// TwinCAT 3 PLC project PLC_InjectionMolding
// ProgramVersion: 3.1.4024.0
// libraries:
//   Tc2_Standard, * (Beckhoff Automation GmbH)
//   Tc2_System, * (Beckhoff Automation GmbH)
//   Tc3_Module, * (Beckhoff Automation GmbH)
//   Tc3_Vision, * (Beckhoff Automation GmbH)
//   VisuDialogs, * (System)
// project tree:
//   DUTs/ ST_ProductionData.TcDUT, E_AlarmID.TcDUT, E_MachineMode.TcDUT, E_SequenceState.TcDUT, ST_Recipe.TcDUT, ST_VisionResult.TcDUT
//   / GlobalTextList.TcGTLO, PlcTask.TcTTO, Visualization Manager.TcVMO (not stored)
//   GVLs/ GVL_Config.TcGVL, GVL_IO.TcGVL, GVL_Simulation.TcGVL, GVL_Status.TcGVL
//   POUs/ FB_AlarmManager.TcPOU, FB_AnalogInput.TcPOU, FB_Extruder.TcPOU, FB_Hopper.TcPOU, FB_InjectionSequence.TcPOU, FB_Interlocks.TcPOU, FB_Machine.TcPOU, FB_Mold.TcPOU, FB_PlantSimulation.TcPOU, FB_TemperatureControl.TcPOU, FB_Vision.TcPOU, MAIN.TcPOU, PRG_VisionTest.TcPOU
//   VISUs/ Visualization_Overview.TcVIS
// real-time tasks:
//   TASK PlcTask: cycle T#10ms, priority 20, ADS port 350

CONFIGURATION PLC_InjectionMolding
    RESOURCE PLC ON TwinCAT3
        TASK PlcTask(INTERVAL := T#10ms, PRIORITY := 20);
        PROGRAM MAIN WITH PlcTask : MAIN;
        PROGRAM PRG_VisionTest WITH PlcTask : PRG_VisionTest;
    END_RESOURCE
END_CONFIGURATION

// ---- DUTs/ST_ProductionData.TcDUT
TYPE ST_ProductionData :
STRUCT
	nTotalParts        : UDINT;
    nGoodParts         : UDINT;
    nRejectedParts     : UDINT;

    fRejectRate        : REAL;

    tLastCycleTime     : TIME;

    nLastDefectCode    : UINT;
	
	fLastCycleTimeSec : REAL;
END_STRUCT
END_TYPE

// ---- DUTs/E_AlarmID.TcDUT
{attribute 'qualified_only'}
{attribute 'strict'}
TYPE E_AlarmID :
(
	ALARM_NONE:=0,
	
	//HOPPER
	ALARM_HOPPER_LOW_TIMEOUT:=1001,
	ALARM_HOPPER_FILL_TIMEOUT:=1002,
	
	//TEMPERATURE/PRESSURE
	ALARM_TEMP_LOW:=2001,
	ALARM_TEMP_HIGH:=2002,
	ALARM_PRESSURE_HIGH:=2003,
	
	//MOLD/MOTION
	ALARM_MOLD_OPEN_TIMEOUT:=3001,
	ALARM_MOLD_CLOSE_TIMEOUT:=3002,
	
	//VISION
	ALARM_VISION_OFFLINE:=4001,
	ALARM_VISION_TIMEOUT:=4002,
	
	//SAFETY
	ALARM_GUARD_OPEN:=9001,
	ALARM_ESTOP:=9002
);
END_TYPE

// ---- DUTs/E_MachineMode.TcDUT
{attribute 'qualified_only'}
{attribute 'strict'}
TYPE E_MachineMode :
(
	MODE_INITIAL := 0,
    MODE_STARTUP := 1,
    MODE_STOPPED := 2,
    MODE_RUN := 3,
    MODE_SHUTDOWN := 4,
    MODE_ESTOP := 5	
);
END_TYPE

// ---- DUTs/E_SequenceState.TcDUT
{attribute 'qualified_only'}
{attribute 'strict'}
TYPE E_SequenceState :
(
	SEQ_IDLE :=0,
	SEQ_INJECT :=1,
	SEQ_COOLING :=2,
	SEQ_DOSING :=3,
	SEQ_OPEN_MOLD :=4,
	SEQ_EJECT:=5,
	SEQ_CLOSE_MOLD:=6,
	
	//Vision
	SEQ_VISION_TRIGGER:=7,
	SEQ_VISION_WAIT:=8,
	SEQ_SORT_PART:=9,
	
	SEQ_COMPLETE:= 10
);
END_TYPE

// ---- DUTs/ST_Recipe.TcDUT
TYPE ST_Recipe :
STRUCT
	sProductName		: STRING(40);
	
	fBarrelTempSP       : REAL;
    fPressureLimit      : REAL;

    tCoolingTime        : TIME;
    tInjectionTimeout   : TIME;

    nVisionJob          : UINT;

    fWidthMin           : REAL;
    fWidthMax           : REAL;
    fHeightMin          : REAL;
    fHeightMax          : REAL;
	
END_STRUCT
END_TYPE

// ---- DUTs/ST_VisionResult.TcDUT
TYPE ST_VisionResult :
STRUCT

    // Vision system status
    bReady       : BOOL;
    bBusy        : BOOL;

    // Result handshake
    bResultValid : BOOL;

    // Inspection result
    bPartPresent : BOOL;
    bPartOK      : BOOL;

    // Classification
    nDefectCode  : UINT;

    // Measured geometry
    // Currently stored in pixels
    fWidth       : REAL;
    fHeight      : REAL;
    fAngle       : REAL;

    // Identification of inspected part
    nProductID   : DINT;

END_STRUCT
END_TYPE

// ---- GVLs/GVL_Config.TcGVL
{attribute 'qualified_only'}
VAR_GLOBAL
	// Temperature Configuration
	
	c_fStartupTempSP      : REAL := 120.0;
    c_fShutdownTempSP     : REAL := 20.0;
    c_fShutdownComplete   : REAL := 30.0;
	
	// Pressure Limits
	
	c_fStartupPressure    : REAL := 4.0;
    c_fMaxPressure        : REAL := 100.0;
	c_fMinOperatingTemp	  : REAL := 80.0;
	
	// Process Timing
	
	c_tCoolingTime        : TIME := T#5S;
	
	// Hopper Monitoring
	
	c_tHopperLowTimeout   : TIME := T#30S;
    c_tHopperFillTimeout  : TIME := T#180S;
	
	// Production
	
	c_nBatchSize          : UDINT := 1000;	
	
END_VAR

// ---- GVLs/GVL_IO.TcGVL
{attribute 'qualified_only'}
VAR_GLOBAL
	
	//Operator Inputs
	
	B_start		: BOOL;
	B_ES		: BOOL;
	B_ack		: BOOL;
	B_startup	: BOOL;
	B_shutdown	: BOOL;
	B_stop		: BOOL;
	
	//Position Sensors
	
	ES101		: BOOL;
	ES102		: BOOL;
	ES201		: BOOL;
	ES202		: BOOL;
	
	//Safety
	
	S101		: BOOL;
	
	//Hopper Sensors
	
	LIS101		: BOOL;
	LIS102		: BOOL;	
	
	//Analog Inputs
	
	PI101_raw	: INT;
	TI101_raw	: INT;
	TI201_raw	: INT;
	
	//Motors
	
	M101         : BOOL;
    M102         : BOOL;
    M201_l       : BOOL;
    M201_r       : BOOL;
    M301         : BOOL;
	
	//Valves
	
	V1           : BOOL;
    V2           : BOOL;
    V3           : BOOL;
	
	//Heating
	
	P_in		 : REAL;
	
	//Hopper Warning
	
	W_hopper	 : BOOL;
	
END_VAR

// ---- GVLs/GVL_Simulation.TcGVL
{attribute 'qualified_only'}

VAR_GLOBAL

    // =====================================================
    // MASTER SWITCH
    // =====================================================

    bSimulationEnabled : BOOL := TRUE;


    // =====================================================
    // FAULT INJECTION
    // =====================================================

    bForcePressureHigh : BOOL := FALSE;
    bForceTempLow      : BOOL := FALSE;

    bForceES101Fault   : BOOL := FALSE;
    bForceES102Fault   : BOOL := FALSE;
    bForceES201Fault   : BOOL := FALSE;
    bForceES202Fault   : BOOL := FALSE;

    bForceLIS101Fault  : BOOL := FALSE;
    bForceLIS102Fault  : BOOL := FALSE;


    // =====================================================
    // VISION FAULT INJECTION
    // =====================================================

    bForceVisionOffline : BOOL := FALSE;

    // Kept for compatibility / old commissioning logic.
    // The new FB_Vision does not need this for real defect detection.
    bForceVisionReject  : BOOL := FALSE;

    bForceVisionTimeout : BOOL := FALSE;


    // =====================================================
    // VISION IMAGE SOURCE
    // =====================================================

    // Used by FB_Vision.
    // In manual mode, set this directly.
    // In random mode, MAIN updates it automatically.
    sVisionImagePath : STRING(255) :=
        'C:\TcVision\good_reference.png';


    // =====================================================
    // RANDOM VIRTUAL PART MODE
    // =====================================================

    // FALSE = manually choose sVisionImagePath
    // TRUE  = randomly select one dataset image
    //         whenever a new part enters SEQ_INJECT
    bRandomPartMode : BOOL := TRUE;


    // Current image selected for the molded part
    nVisionDatasetIndex : INT := 1;


    // Seed for pseudo-random number generator
    // Fixed value makes the sequence reproducible
    nRandomSeed : UDINT := 123456789;


    // =====================================================
    // RANDOM VISION DATASET
    // =====================================================

    aVisionDataset : ARRAY[1..40] OF STRING(255) := [

        'C:\TcVision\RandomDataset\part_001.png',
        'C:\TcVision\RandomDataset\part_002.png',
        'C:\TcVision\RandomDataset\part_003.png',
        'C:\TcVision\RandomDataset\part_004.png',
        'C:\TcVision\RandomDataset\part_005.png',
        'C:\TcVision\RandomDataset\part_006.png',
        'C:\TcVision\RandomDataset\part_007.png',
        'C:\TcVision\RandomDataset\part_008.png',
        'C:\TcVision\RandomDataset\part_009.png',
        'C:\TcVision\RandomDataset\part_010.png',

        'C:\TcVision\RandomDataset\part_011.png',
        'C:\TcVision\RandomDataset\part_012.png',
        'C:\TcVision\RandomDataset\part_013.png',
        'C:\TcVision\RandomDataset\part_014.png',
        'C:\TcVision\RandomDataset\part_015.png',
        'C:\TcVision\RandomDataset\part_016.png',
        'C:\TcVision\RandomDataset\part_017.png',
        'C:\TcVision\RandomDataset\part_018.png',
        'C:\TcVision\RandomDataset\part_019.png',
        'C:\TcVision\RandomDataset\part_020.png',

        'C:\TcVision\RandomDataset\part_021.png',
        'C:\TcVision\RandomDataset\part_022.png',
        'C:\TcVision\RandomDataset\part_023.png',
        'C:\TcVision\RandomDataset\part_024.png',
        'C:\TcVision\RandomDataset\part_025.png',
        'C:\TcVision\RandomDataset\part_026.png',
        'C:\TcVision\RandomDataset\part_027.png',
        'C:\TcVision\RandomDataset\part_028.png',
        'C:\TcVision\RandomDataset\part_029.png',
        'C:\TcVision\RandomDataset\part_030.png',

        'C:\TcVision\RandomDataset\part_031.png',
        'C:\TcVision\RandomDataset\part_032.png',
        'C:\TcVision\RandomDataset\part_033.png',
        'C:\TcVision\RandomDataset\part_034.png',
        'C:\TcVision\RandomDataset\part_035.png',
        'C:\TcVision\RandomDataset\part_036.png',
        'C:\TcVision\RandomDataset\part_037.png',
        'C:\TcVision\RandomDataset\part_038.png',
        'C:\TcVision\RandomDataset\part_039.png',
        'C:\TcVision\RandomDataset\part_040.png'

    ];

END_VAR

// ---- GVLs/GVL_Status.TcGVL
{attribute 'qualified_only'}
VAR_GLOBAL
	

	eMachineMode:
		E_MachineMode:= E_MachineMode.MODE_INITIAL;
		
	eSequenceState:
		E_SequenceState:= E_SequenceState.SEQ_IDLE;
		
	stProduction:
		ST_ProductionData;
		
	stVision:
		ST_VisionResult;
		
	//Process Values
	
	fPressureBar      : REAL := 0.0;
    fBarrelTemp       : REAL := 20.0;
    fMoldTemp         : REAL := 20.0;

	//Machine Status

	bMachineReady     : BOOL := FALSE;
    bCycleActive      : BOOL := FALSE;
    bFaultActive      : BOOL := FALSE;	
	
	eActiveAlarm : E_AlarmID := E_AlarmID.ALARM_NONE;
	sSequenceText : STRING(32) := 'IDLE';
	sMachineModeText : STRING(20) := 'INITIAL';
	sActiveAlarmText : STRING(40) := 'NONE';
END_VAR

// ---- POUs/MAIN.TcPOU
PROGRAM MAIN
VAR
	fbPlantSim   : FB_PlantSimulation;

    fbPressure   : FB_AnalogInput;
    fbBarrelTemp : FB_AnalogInput;
    fbMoldTemp   : FB_AnalogInput;
	fbMachine	 : FB_Machine;
	fbTemperature: FB_TemperatureControl;
	fbInjectionSequence : FB_InjectionSequence;
	fbExtruder	 : FB_Extruder;
	fbMold		 : FB_Mold;
	fbHopper	 : FB_Hopper;
	fbAlarmManager : FB_AlarmManager;
	fbInterlocks : FB_Interlocks;

	// Temporary manual commands for commissioning/testing
	bTestM101_Request   : BOOL := FALSE;
	bTestM102_Request   : BOOL := FALSE;
	bTestM201_l_Request : BOOL := FALSE;
	bTestM201_r_Request : BOOL := FALSE;
	
	 // Vision
    fbVision              : FB_Vision;
    bVisionTestTrigger    : BOOL := FALSE;
    bVisionTestAck        : BOOL := FALSE;
    nVisionTestProductID  : DINT := 1;
    bVisionOffline        : BOOL := FALSE;
	bVisionTimeout : BOOL;
	
	
	nRandomValue : UDINT;
	
	ePreviousSequenceState : E_SequenceState := E_SequenceState.SEQ_IDLE;
	
END_VAR

										// ANALOG INPUT PROCESSING


// Pressure PI101: 0 ... 200 bar
fbPressure(
    nRaw := GVL_IO.PI101_raw,
    fEngMin := 0.0,
    fEngMax := 200.0,
    fValue => GVL_Status.fPressureBar
);


// Barrel temperature TI101: -100 ... 600 °C
fbBarrelTemp(
    nRaw := GVL_IO.TI101_raw,
    fEngMin := -100.0,
    fEngMax := 600.0,
    fValue => GVL_Status.fBarrelTemp
);


// Mold temperature TI201: -100 ... 600 °C
fbMoldTemp(
    nRaw := GVL_IO.TI201_raw,
    fEngMin := -100.0,
    fEngMax := 600.0,
    fValue => GVL_Status.fMoldTemp
);

														// MACHINE MODE CONTROL

fbMachine(
    bStartup := GVL_IO.B_startup,
    bStart := GVL_IO.B_start,
    bStop := GVL_IO.B_stop,
    bShutdown := GVL_IO.B_shutdown,
    bEStop := GVL_IO.B_ES,
    bAck := GVL_IO.B_ack,

    fBarrelTemp := GVL_Status.fBarrelTemp,
    fPressureBar := GVL_Status.fPressureBar,
    bMoldClosed := GVL_IO.ES202,

    bSequenceStopComplete :=
        fbInjectionSequence.bStopComplete,

    eMode => GVL_Status.eMachineMode,
    bMachineReady => GVL_Status.bMachineReady,

    bV2 => GVL_IO.V2,
    bV3 => GVL_IO.V3
);


														// TEMPERATURE CONTROL
fbTemperature(
    bEnable := fbMachine.bTempControlEnable,
	fSetpoint := fbMachine.fTempSetpoint,
    fActualTemp := GVL_Status.fBarrelTemp,

    fHeatingPower => GVL_IO.P_in,
    bCoolingValve => GVL_IO.V1
);

													// AUTOMATIC INJECTION SEQUENCE


fbInjectionSequence(
    bEnable :=
        GVL_Status.eMachineMode =
        E_MachineMode.MODE_RUN,

    bStopRequest := GVL_IO.B_stop,

    bAtFront := GVL_IO.ES101,
    bAtRear := GVL_IO.ES102,

    bMoldOpen := GVL_IO.ES201,
    bMoldClosed := GVL_IO.ES202,

    tCoolingTime := GVL_Config.c_tCoolingTime,

    nProducedParts :=
        GVL_Status.stProduction.nTotalParts,

    nBatchSize :=
        GVL_Config.c_nBatchSize,
		
	bVisionReady :=
    	GVL_Status.stVision.bReady,

	bVisionResultValid :=
    	GVL_Status.stVision.bResultValid,

	bVisionPartOK :=
    	GVL_Status.stVision.bPartOK,
		
	bVisionOffline := fbVision.bOffline,

	bVisionTimeout := fbVision.bTimeout,

    eState => GVL_Status.eSequenceState,
	
	tLastCycleTime =>
        GVL_Status.stProduction.tLastCycleTime
);

	GVL_Status.bCycleActive := fbInjectionSequence.bCycleActive;
	
	GVL_Status.stProduction.fLastCycleTimeSec :=
    	TIME_TO_REAL(GVL_Status.stProduction.tLastCycleTime) / 1000.0;
	

CASE GVL_Status.eMachineMode OF

    E_MachineMode.MODE_INITIAL:
        GVL_Status.sMachineModeText := 'INITIAL';

    E_MachineMode.MODE_STARTUP:
        GVL_Status.sMachineModeText := 'STARTUP';

    E_MachineMode.MODE_STOPPED:
        GVL_Status.sMachineModeText := 'STOPPED';

    E_MachineMode.MODE_RUN:
        GVL_Status.sMachineModeText := 'RUN';

    E_MachineMode.MODE_SHUTDOWN:
        GVL_Status.sMachineModeText := 'SHUTDOWN';

    E_MachineMode.MODE_ESTOP:
        GVL_Status.sMachineModeText := 'E-STOP';

ELSE
    GVL_Status.sMachineModeText := 'UNKNOWN';

END_CASE;





CASE fbInjectionSequence.eState OF

    E_SequenceState.SEQ_IDLE:
        GVL_Status.sSequenceText := 'IDLE';

    E_SequenceState.SEQ_INJECT:
        GVL_Status.sSequenceText := 'INJECT';

    E_SequenceState.SEQ_COOLING:
        GVL_Status.sSequenceText := 'COOLING';

    E_SequenceState.SEQ_DOSING:
        GVL_Status.sSequenceText := 'DOSING';

    E_SequenceState.SEQ_OPEN_MOLD:
        GVL_Status.sSequenceText := 'OPEN MOLD';

    E_SequenceState.SEQ_EJECT:
        GVL_Status.sSequenceText := 'EJECT';

    E_SequenceState.SEQ_CLOSE_MOLD:
        GVL_Status.sSequenceText := 'CLOSE MOLD';

    E_SequenceState.SEQ_VISION_TRIGGER:
        GVL_Status.sSequenceText := 'VISION TRIGGER';

    E_SequenceState.SEQ_VISION_WAIT:
        GVL_Status.sSequenceText := 'VISION WAIT';

    E_SequenceState.SEQ_SORT_PART:
        GVL_Status.sSequenceText := 'SORT PART';

    E_SequenceState.SEQ_COMPLETE:
        GVL_Status.sSequenceText := 'COMPLETE';

ELSE
    GVL_Status.sSequenceText := 'UNKNOWN';

END_CASE;



// =====================================================
// RANDOM VIRTUAL PART GENERATOR
// Select exactly one image when a new cycle enters
// SEQ_INJECT.
// =====================================================

IF GVL_Simulation.bRandomPartMode
   AND
   (fbInjectionSequence.eState = E_SequenceState.SEQ_INJECT)
   AND
   (ePreviousSequenceState <> E_SequenceState.SEQ_INJECT) THEN

    // -------------------------------------------------
    // Generate next pseudo-random number
    // -------------------------------------------------

    GVL_Simulation.nRandomSeed :=
        (GVL_Simulation.nRandomSeed * UDINT#1664525)
        + UDINT#1013904223;

    nRandomValue :=
        GVL_Simulation.nRandomSeed;


    // -------------------------------------------------
    // Map pseudo-random value to dataset index 1..40
    // -------------------------------------------------

    GVL_Simulation.nVisionDatasetIndex :=
        UDINT_TO_INT(
            nRandomValue MOD UDINT#40
        ) + 1;


    // -------------------------------------------------
    // Assign selected image to this molded part
    // -------------------------------------------------

    GVL_Simulation.sVisionImagePath :=
        GVL_Simulation.aVisionDataset[
            GVL_Simulation.nVisionDatasetIndex
        ];

END_IF;


// =====================================================
// STORE CURRENT STATE FOR NEXT PLC SCAN
// This line MUST come after the random-selection logic.
// =====================================================

ePreviousSequenceState :=
    fbInjectionSequence.eState;	
	
	
	
	
											// COUNT PRODUCED PARTS

IF fbInjectionSequence.bPartCompleted THEN

    GVL_Status.stProduction.nTotalParts :=
        GVL_Status.stProduction.nTotalParts + 1;

END_IF;

// Good part counter
IF fbInjectionSequence.bGoodPart THEN

    GVL_Status.stProduction.nGoodParts :=
        GVL_Status.stProduction.nGoodParts + 1;

END_IF;


// Rejected part counter
IF fbInjectionSequence.bRejectedPart THEN

    GVL_Status.stProduction.nRejectedParts :=
        GVL_Status.stProduction.nRejectedParts + 1;

    // Store meaningful reject reason
    IF fbVision.bOffline THEN

        // Vision system unavailable
        GVL_Status.stProduction.nLastDefectCode := UINT#4001;

    ELSIF fbVision.bTimeout THEN

        // Vision inspection timeout
        GVL_Status.stProduction.nLastDefectCode := UINT#4002;

    ELSE

        // Genuine Cognex / simulated inspection defect
        GVL_Status.stProduction.nLastDefectCode :=
            GVL_Status.stVision.nDefectCode;

    END_IF;

END_IF;


// Reject rate
IF GVL_Status.stProduction.nTotalParts > 0 THEN

    GVL_Status.stProduction.fRejectRate :=
        (
            UDINT_TO_REAL(
                GVL_Status.stProduction.nRejectedParts
            )
            /
            UDINT_TO_REAL(
                GVL_Status.stProduction.nTotalParts
            )
        ) * 100.0;

ELSE

    GVL_Status.stProduction.fRejectRate := 0.0;

END_IF;


											// EQUIPMENT CONTROL (Extruder + MOLD)

fbExtruder(
    bRotateCmd :=
        fbMachine.bStartupRotateCmd
        OR fbInjectionSequence.bRotateCmd,

    bInjectCmd :=
        fbInjectionSequence.bInjectCmd,

    bES101 := GVL_IO.ES101,
    bES102 := GVL_IO.ES102
);

fbMold(
    bOpenCmd :=
        fbInjectionSequence.bOpenMoldCmd,

    bCloseCmd :=
        fbMachine.bStartupCloseCmd
        OR fbInjectionSequence.bCloseMoldCmd,

    bES201 := GVL_IO.ES201,
    bES202 := GVL_IO.ES202
);

										// MACHINE INTERLOCKS

fbInterlocks(
    eMode := GVL_Status.eMachineMode,
	bM101_Request := fbExtruder.bRotateRequest,
    bM102_Request := fbExtruder.bInjectRequest,
    bM201_l_Request := fbMold.bOpenRequest,
    bM201_r_Request := fbMold.bCloseRequest,

    bES101 := GVL_IO.ES101,
    bES102 := GVL_IO.ES102,
    bES201 := GVL_IO.ES201,
    bES202 := GVL_IO.ES202,

    bGuardOpen := GVL_IO.S101,

    fPressureBar := GVL_Status.fPressureBar,
    fBarrelTemp := GVL_Status.fBarrelTemp,

    bM101_Enable => GVL_IO.M101,
    bM102_Enable => GVL_IO.M102,
    bM201_l_Enable => GVL_IO.M201_l,
    bM201_r_Enable => GVL_IO.M201_r
);

																	// HOPPER CONTROL

fbHopper(
    eMode := GVL_Status.eMachineMode,

    bLIS101 := GVL_IO.LIS101,
    bLIS102 := GVL_IO.LIS102,

    bAck := GVL_IO.B_ack,

    bFeederRequest => GVL_IO.M301,
    bWarning => GVL_IO.W_hopper
);


// =====================================================
// RANDOM VIRTUAL PART GENERATOR
// Select one image exactly once when entering SEQ_INJECT
// =====================================================

IF GVL_Simulation.bRandomPartMode
   AND
   (fbInjectionSequence.eState = E_SequenceState.SEQ_INJECT)
   AND
   (ePreviousSequenceState <> E_SequenceState.SEQ_INJECT) THEN

    // Generate next pseudo-random number
    GVL_Simulation.nRandomSeed :=
        (GVL_Simulation.nRandomSeed * UDINT#1664525)
        + UDINT#1013904223;

    nRandomValue :=
        GVL_Simulation.nRandomSeed;


    // Convert random value to dataset index 1..40
    GVL_Simulation.nVisionDatasetIndex :=
        UDINT_TO_INT(
            nRandomValue MOD UDINT#40
        ) + 1;


    // Assign selected image to current molded part
    GVL_Simulation.sVisionImagePath :=
        GVL_Simulation.aVisionDataset[
            GVL_Simulation.nVisionDatasetIndex
        ];

END_IF;


// IMPORTANT:
// Store current state only AFTER the random selection check
ePreviousSequenceState :=
    fbInjectionSequence.eState;



																	// VISION SYSTEM
// Temporary simulation / commissioning interface

fbVision(
    bEnable :=
        (GVL_Status.eMachineMode = E_MachineMode.MODE_RUN),

    bTrigger :=
        fbInjectionSequence.bVisionTrigger,

    bAck :=
        fbInjectionSequence.bVisionAck,

    bFaultAck :=
        GVL_IO.B_ack,

    bForceOffline :=
        GVL_Simulation.bForceVisionOffline,

    bForceTimeout :=
        GVL_Simulation.bForceVisionTimeout,

    nProductID :=
        UDINT_TO_DINT(
            GVL_Status.stProduction.nTotalParts + 1
        ),
		
	sImagePath :=
		GVL_Simulation.sVisionImagePath,

    stResult =>
        GVL_Status.stVision,

    bOffline =>
        bVisionOffline,
		
	bTimeout =>
        bVisionTimeout
);

																	// ALARM MANAGEMENT


fbAlarmManager(
    eMode := GVL_Status.eMachineMode,

    bHopperLowTimeout :=
        fbHopper.bLowLevelTimeout,

    bHopperFillTimeout :=
        fbHopper.bFillTimeout,

    fBarrelTemp :=
        GVL_Status.fBarrelTemp,

    fPressureBar :=
        GVL_Status.fPressureBar,

    bGuardOpen :=
        GVL_IO.S101,

    bEStop :=
        GVL_IO.B_ES,

    bVisionOffline :=
        bVisionOffline,

    bVisionTimeout :=
		fbVision.bTimeout,

    bAck :=
        GVL_IO.B_ack,

    bFaultActive =>
        GVL_Status.bFaultActive,

    eActiveAlarm =>
        GVL_Status.eActiveAlarm
);

CASE GVL_Status.eActiveAlarm OF

    E_AlarmID.ALARM_NONE:
        GVL_Status.sActiveAlarmText := 'NONE';

    E_AlarmID.ALARM_VISION_OFFLINE:
        GVL_Status.sActiveAlarmText := 'VISION OFFLINE';

    E_AlarmID.ALARM_VISION_TIMEOUT:
        GVL_Status.sActiveAlarmText := 'VISION TIMEOUT';

ELSE
    GVL_Status.sActiveAlarmText := 'ALARM ACTIVE';

END_CASE;

											// PLANT SIMULATION

fbPlantSim(
    bEnable := GVL_Simulation.bSimulationEnabled,

    bM101 := GVL_IO.M101,
    bM102 := GVL_IO.M102,
    bM201_l := GVL_IO.M201_l,
    bM201_r := GVL_IO.M201_r,
    bM301 := GVL_IO.M301,

    bV1 := GVL_IO.V1,
    bV2 := GVL_IO.V2,
    bV3 := GVL_IO.V3,

    fHeaterPower := GVL_IO.P_in,

    eMode := GVL_Status.eMachineMode,

    bES101 => GVL_IO.ES101,
    bES102 => GVL_IO.ES102,
    bES201 => GVL_IO.ES201,
    bES202 => GVL_IO.ES202,

    bLIS101 => GVL_IO.LIS101,
    bLIS102 => GVL_IO.LIS102,

    nPI101Raw => GVL_IO.PI101_raw,
    nTI101Raw => GVL_IO.TI101_raw,
    nTI201Raw => GVL_IO.TI201_raw
);

//PRG_VisionTest();

END_PROGRAM

// ---- POUs/FB_PlantSimulation.TcPOU
FUNCTION_BLOCK FB_PlantSimulation
VAR_INPUT
	bEnable		: BOOL;
	
	//Motors
	
	bM101		: BOOL;
	bM102		: BOOL;
	bM201_l		: BOOL;
	bM201_r		: BOOL;
	bM301		: BOOL;
	
	// Valves
	bV1			: BOOL;
	bV2			: BOOL;
	bV3			: BOOL;
	
	// Heater
	fHeaterPower: REAL;
	
	//machine Operating Mode
	eMode		: E_MachineMode;	
END_VAR
VAR_OUTPUT
	// Screw end switches
    bES101        : BOOL;
    bES102        : BOOL;

    // Mold end switches
    bES201        : BOOL;
    bES202        : BOOL;

    // Hopper level switches
    bLIS101       : BOOL;
    bLIS102       : BOOL;

    // Simulated analog inputs
    nPI101Raw     : INT;
    nTI101Raw     : INT;
    nTI201Raw     : INT;
END_VAR
VAR
	 // Positions: 0 ... 100 %
    fScrewPosition : REAL := 50.0;
    fMoldPosition  : REAL := 0.0;
    fHopperLevel   : REAL := 75.0;

    // Physical process values
    fPressure      : REAL := 0.0;
    fBarrelTemp    : REAL := 20.0;
    fMoldTemp      : REAL := 20.0;
END_VAR

IF bEnable THEN

    									// Injection screw simulation

    // Injection cylinder pushes screw forward
    IF bM102 THEN
        fScrewPosition := fScrewPosition + 1.0;
    END_IF;


    // During normal operation M101 performs dosing,
    // causing the screw to move backwards.
    IF bM101 AND
       (eMode = E_MachineMode.MODE_RUN) THEN

        fScrewPosition := fScrewPosition - 0.5;

    END_IF;


    // Limit screw position
    fScrewPosition :=
        LIMIT(0.0, fScrewPosition, 100.0);


    // Generate end switches
    bES101 := (fScrewPosition >= 100.0);
    bES102 := (fScrewPosition <= 0.0);



   
    											// Mold simulation
  

    IF bM201_l THEN
        fMoldPosition := fMoldPosition - 0.2;
    END_IF;

    IF bM201_r THEN
        fMoldPosition := fMoldPosition + 0.2;
    END_IF;


    fMoldPosition :=
        LIMIT(0.0, fMoldPosition, 100.0);


    bES201 := (fMoldPosition <= 0.0);
    bES202 := (fMoldPosition >= 100.0);

	
    										 // Hopper simulation
											 

    IF bM301 THEN

        fHopperLevel := fHopperLevel + 0.05;

    ELSIF eMode = E_MachineMode.MODE_RUN THEN

        // Material consumption
        fHopperLevel := fHopperLevel - 0.002;

    END_IF;


    fHopperLevel :=
        LIMIT(0.0, fHopperLevel, 100.0);


    // Low-level sensor
    //bLIS101 := (fHopperLevel > 20.0);

    // High-level sensor
    //bLIS102 := (fHopperLevel >= 90.0);
	
	// Normal level-switch simulation
	bLIS101 := (fHopperLevel > 20.0);
	bLIS102 := (fHopperLevel >= 90.0);

	// Fault injection
	IF GVL_Simulation.bForceLIS101Fault THEN
    	bLIS101 := FALSE;
	END_IF;

	IF GVL_Simulation.bForceLIS102Fault THEN
    	bLIS102 := FALSE;
	END_IF;



    									// Barrel Temperature Simulation

    IF fHeaterPower > 0.0 THEN

        fBarrelTemp :=
            fBarrelTemp +
            (fHeaterPower / 100.0) * 0.03;

    END_IF;


    // Cooling valve
    IF bV1 THEN
        fBarrelTemp := fBarrelTemp - 0.02;
    END_IF;


    // Natural cooling toward ambient
    IF (fHeaterPower <= 0.0) AND NOT bV1 THEN

        IF fBarrelTemp > 20.0 THEN
            fBarrelTemp := fBarrelTemp - 0.002;
        END_IF;

    END_IF;


    fBarrelTemp :=
        LIMIT(-100.0, fBarrelTemp, 600.0);


										   // Mold Temperature Simulation

    IF bV2 OR bV3 THEN

        IF fMoldTemp > 20.0 THEN
            fMoldTemp := fMoldTemp - 0.01;
        END_IF;

    END_IF;


    fMoldTemp :=
        LIMIT(-100.0, fMoldTemp, 600.0);


										    // Pressure Simulation
 

// During startup, screw rotation fills the nozzle
// and pressure gradually rises.
IF eMode = E_MachineMode.MODE_STARTUP THEN

    IF bM101 THEN
        fPressure := fPressure + 0.01;
    END_IF;


// During normal production
ELSIF eMode = E_MachineMode.MODE_RUN THEN

    // Injection temporarily raises pressure
    IF bM102 THEN

        fPressure := fPressure + 0.10;

    ELSE

        // Pressure relaxes after injection
        IF fPressure > 5.0 THEN
            fPressure := fPressure - 0.10;

        ELSIF fPressure < 5.0 THEN
            fPressure := fPressure + 0.01;
        END_IF;

    END_IF;


// Machine not producing
ELSE

    IF fPressure > 0.0 THEN
        fPressure := fPressure - 0.05;
    END_IF;

END_IF;


// Physical limits
fPressure :=
    LIMIT(0.0, fPressure, 200.0);

						    // Convert physical values back to raw PLC signals
 
    nPI101Raw :=
        REAL_TO_INT(
            (fPressure / 200.0) * 32767.0
        );


    nTI101Raw :=
        REAL_TO_INT(
            ((fBarrelTemp + 100.0) / 700.0)
            * 32767.0
        );


    nTI201Raw :=
        REAL_TO_INT(
            ((fMoldTemp + 100.0) / 700.0)
            * 32767.0
        );

END_IF;

END_FUNCTION_BLOCK

// ---- POUs/FB_AnalogInput.TcPOU
FUNCTION_BLOCK FB_AnalogInput
VAR_INPUT
	nRaw	:	INT;
	fEngMin :	REAL;
	fEngMax :	REAL;
END_VAR

VAR_OUTPUT
	fValue  :	REAL;
	bValid  :	BOOL;
END_VAR

VAR
	fRaw	:	REAL;
END_VAR

fRaw:= INT_TO_REAL(nRaw);

bValid := (nRaw >= 0);

IF bValid THEN
	fValue := fEngMin+(fRaw/32768.0)*(fEngMax -fEngMin);
ELSE
	fValue := fEngMin;
END_IF

END_FUNCTION_BLOCK

// ---- POUs/FB_Machine.TcPOU
FUNCTION_BLOCK FB_Machine
VAR_INPUT
    // Operator controls
    bStartup        : BOOL;
    bStart          : BOOL;
    bStop           : BOOL;
    bShutdown       : BOOL;
    bEStop          : BOOL;
    bAck            : BOOL;

    // Process feedback
    fBarrelTemp     : REAL;
    fPressureBar    : REAL;
    bMoldClosed     : BOOL;

    // Sequence feedback
    bSequenceStopComplete : BOOL;
END_VAR

VAR_OUTPUT
    eMode               : E_MachineMode := E_MachineMode.MODE_INITIAL;

    // Temperature system
    bTempControlEnable  : BOOL;
    fTempSetpoint       : REAL;

    // Mold cooling
    bV2                 : BOOL;
    bV3                 : BOOL;

    // Startup commands
    bStartupRotateCmd   : BOOL;
    bStartupCloseCmd    : BOOL;

    // Status
    bMachineReady       : BOOL;
END_VAR

// Default commands every scan
bStartupRotateCmd := FALSE;
bStartupCloseCmd := FALSE;
bMachineReady := FALSE;


// Emergency stop has highest priority

IF bEStop THEN
    eMode := E_MachineMode.MODE_ESTOP;
END_IF;


CASE eMode OF

    // INITIAL

    E_MachineMode.MODE_INITIAL:

        bTempControlEnable := FALSE;
        fTempSetpoint := GVL_Config.c_fShutdownTempSP;

        bV2 := FALSE;
        bV3 := FALSE;

        IF bStartup AND NOT bEStop THEN
            eMode := E_MachineMode.MODE_STARTUP;
        END_IF;

    // STARTUP

    E_MachineMode.MODE_STARTUP:

        bTempControlEnable := TRUE;
        fTempSetpoint := GVL_Config.c_fStartupTempSP;

        bV2 := TRUE;
        bV3 := TRUE;


        // Wait until barrel reaches required temperature
        IF fBarrelTemp >= GVL_Config.c_fStartupTempSP THEN

            // M101 runs until nozzle pressure reaches 4 bar
            IF fPressureBar < GVL_Config.c_fStartupPressure THEN
                bStartupRotateCmd := TRUE;
            END_IF;

            // Mold closes independently
            IF NOT bMoldClosed THEN
                bStartupCloseCmd := TRUE;
            END_IF;


            // Both startup conditions complete
            IF (fPressureBar >= GVL_Config.c_fStartupPressure)
               AND bMoldClosed THEN

                eMode := E_MachineMode.MODE_STOPPED;

            END_IF;

        END_IF;

    // STOPPED / READY

    E_MachineMode.MODE_STOPPED:

        bTempControlEnable := TRUE;
        fTempSetpoint := GVL_Config.c_fStartupTempSP;

        bV2 := TRUE;
        bV3 := TRUE;

        bMachineReady := TRUE;


        IF bStart THEN

            eMode := E_MachineMode.MODE_RUN;

        ELSIF bShutdown THEN

            eMode := E_MachineMode.MODE_SHUTDOWN;

        END_IF;

    // NORMAL PRODUCTION

    E_MachineMode.MODE_RUN:

        bTempControlEnable := TRUE;
        fTempSetpoint := GVL_Config.c_fStartupTempSP;

        bV2 := TRUE;
        bV3 := TRUE;


        // Sequence itself finishes the current part
        // before declaring stop complete.
        IF bSequenceStopComplete THEN
            eMode := E_MachineMode.MODE_STOPPED;
        END_IF;

    // SHUTDOWN

    E_MachineMode.MODE_SHUTDOWN:

        bTempControlEnable := TRUE;
        fTempSetpoint := GVL_Config.c_fShutdownTempSP;

        bV2 := FALSE;
        bV3 := FALSE;


        IF fBarrelTemp <= GVL_Config.c_fShutdownComplete THEN

            bTempControlEnable := FALSE;

            eMode := E_MachineMode.MODE_INITIAL;

        END_IF;

    // EMERGENCY STOP

    E_MachineMode.MODE_ESTOP:

        bTempControlEnable := FALSE;

        bV2 := FALSE;
        bV3 := FALSE;

        bStartupRotateCmd := FALSE;
        bStartupCloseCmd := FALSE;


        IF bAck AND NOT bEStop THEN
            eMode := E_MachineMode.MODE_INITIAL;
        END_IF;


    ELSE

        eMode := E_MachineMode.MODE_INITIAL;

END_CASE;

END_FUNCTION_BLOCK

// ---- POUs/FB_TemperatureControl.TcPOU
FUNCTION_BLOCK FB_TemperatureControl
VAR_INPUT
    bEnable     : BOOL;
    fSetpoint   : REAL;
    fActualTemp : REAL;
END_VAR

VAR_OUTPUT
    fControlOutput : REAL;   // -100 ... +100
    fHeatingPower  : REAL;   // 0 ... 100
    bCoolingValve  : BOOL;

    fError         : REAL;
END_VAR

VAR
    // PID parameters
    fK             : REAL := 100.0;
    fTN            : REAL := 30.0;
    fTV            : REAL := 5.0;

    // Controller states
    fIntegral      : REAL := 0.0;
    fDerivative    : REAL := 0.0;
    fPreviousError : REAL := 0.0;

    // 10 ms PLC task
    fCycleTime     : REAL := 0.01;

    // Cooling PWM
    fCoolingDemand : REAL := 0.0;
    tPWMElapsed    : TIME := T#0MS;
    tPWMOnTime     : TIME := T#0MS;
END_VAR

IF bEnable THEN

    // Control error

    fError := fSetpoint - fActualTemp;

    // Integral term

    fIntegral := fIntegral + (fError * fCycleTime / fTN);

    // Limit integral to avoid excessive wind-up
    fIntegral := LIMIT(-1.0, fIntegral, 1.0);

    // Derivative term

    fDerivative := fTV *(fError - fPreviousError) / fCycleTime;

	 fPreviousError := fError;

    // PID output

    fControlOutput := fK *(fError + fIntegral + fDerivative);

    // Controller output limit
    fControlOutput := LIMIT(-100.0, fControlOutput, 100.0);


ELSE

    fControlOutput := 0.0;
    fIntegral := 0.0;
    fDerivative := 0.0;
    fPreviousError := 0.0;

END_IF;


// Heating

IF fControlOutput > 0.0 THEN

    fHeatingPower := fControlOutput;
    fCoolingDemand := 0.0;

ELSE

    fHeatingPower := 0.0;
    fCoolingDemand := ABS(fControlOutput);

END_IF;

// Cooling PWM Period = 2 seconds

IF bEnable AND (fCoolingDemand > 0.0) THEN

    tPWMElapsed := tPWMElapsed + T#10MS;

    // Restart PWM cycle every 2 seconds
    IF tPWMElapsed >= T#2S THEN
        tPWMElapsed := T#0MS;
    END_IF;


    // Convert percentage to ON duration
    tPWMOnTime :=
        REAL_TO_TIME(
            (fCoolingDemand / 100.0) * 2000.0
        );


    bCoolingValve :=
        tPWMElapsed < tPWMOnTime;

ELSE

    bCoolingValve := FALSE;
    tPWMElapsed := T#0MS;

END_IF;

END_FUNCTION_BLOCK

// ---- POUs/FB_InjectionSequence.TcPOU
FUNCTION_BLOCK FB_InjectionSequence
VAR_INPUT
    bEnable         : BOOL;
    bStopRequest    : BOOL;

    // Screw position
    bAtFront        : BOOL;   // ES101
    bAtRear         : BOOL;   // ES102

    // Mold position
    bMoldOpen       : BOOL;   // ES201
    bMoldClosed     : BOOL;   // ES202

    // Configuration
    tCoolingTime    : TIME;
    nProducedParts  : UDINT;
    nBatchSize      : UDINT;
	
	// Vision system
	bVisionReady       : BOOL;
	bVisionResultValid : BOOL;
	bVisionPartOK      : BOOL;
	bVisionOffline : BOOL;
	bVisionTimeout : BOOL;
END_VAR

VAR_OUTPUT
    eState          : E_SequenceState := E_SequenceState.SEQ_IDLE;

    // Equipment commands
    bRotateCmd      : BOOL;
    bInjectCmd      : BOOL;
    bOpenMoldCmd    : BOOL;
    bCloseMoldCmd   : BOOL;

    // Status
    bCycleActive    : BOOL;
    bPartCompleted  : BOOL;
    bStopComplete   : BOOL;
	
	// Vision handshake
	bVisionTrigger : BOOL;
	bVisionAck     : BOOL;

	// Quality result pulses
	bGoodPart     : BOOL;
	bRejectedPart : BOOL;
	
	// Production statistics
    tLastCycleTime : TIME := T#0MS;
END_VAR

VAR
    fbCoolingTimer  : TON;
	fbCycleTimer : TON;
	
    bStopLatched    : BOOL := FALSE;
	bCycleTiming : BOOL := FALSE;
END_VAR

// =====================================================
// DEFAULT OUTPUTS
// =====================================================

// Mechanical commands are generated by the active state.
// Therefore reset them at the beginning of every PLC scan.

bRotateCmd := FALSE;
bInjectCmd := FALSE;

bOpenMoldCmd := FALSE;
bCloseMoldCmd := FALSE;


// Vision handshake outputs are one-scan pulses.

bVisionTrigger := FALSE;
bVisionAck := FALSE;


// Production event outputs are also one-scan pulses.

bPartCompleted := FALSE;
bGoodPart := FALSE;
bRejectedPart := FALSE;

bStopComplete := FALSE;


// Sequence is considered active whenever RUN enables it.

bCycleActive := bEnable;


// =====================================================
// STOP REQUEST LATCH
// =====================================================

// Do not stop immediately.
// Remember the request and finish the current part first.

IF bEnable AND bStopRequest THEN
    bStopLatched := TRUE;
END_IF;


// Batch production complete

IF bEnable
   AND (nProducedParts >= nBatchSize) THEN

    bStopLatched := TRUE;

END_IF;


// =====================================================
// COOLING TIMER
// =====================================================

fbCoolingTimer(
    IN := (eState = E_SequenceState.SEQ_COOLING),
    PT := tCoolingTime
);

// =====================================================
// CYCLE TIME MEASUREMENT
// =====================================================

fbCycleTimer(
    IN := bCycleTiming,
    PT := T#24H
);

// =====================================================
// SEQUENCE DISABLED
// =====================================================

IF NOT bEnable THEN

    eState := E_SequenceState.SEQ_IDLE;

    bStopLatched := FALSE;
	bCycleTiming := FALSE;


// =====================================================
// AUTOMATIC PRODUCTION SEQUENCE
// =====================================================

ELSE

    CASE eState OF


        // -------------------------------------------------
        // IDLE
        // -------------------------------------------------

        E_SequenceState.SEQ_IDLE:

            // Always begin with the mold closed.

            IF NOT bMoldClosed THEN

                bCloseMoldCmd := TRUE;


            // A stop may already have been requested.

            ELSIF bStopLatched THEN

                bStopComplete := TRUE;


            // Machine is ready to produce the next part.

            ELSE

                // Start a new production cycle
    			bCycleTiming := TRUE;
				eState := E_SequenceState.SEQ_INJECT;

            END_IF;



        // -------------------------------------------------
        // INJECTION
        // -------------------------------------------------

        E_SequenceState.SEQ_INJECT:

            bInjectCmd := TRUE;

            // Injection continues until the screw reaches
            // the front end position.

            IF bAtFront THEN

                bInjectCmd := FALSE;

                eState := E_SequenceState.SEQ_COOLING;

            END_IF;



        // -------------------------------------------------
        // COOLING
        // -------------------------------------------------

        E_SequenceState.SEQ_COOLING:

            // fbCoolingTimer runs while this state is active.

            IF fbCoolingTimer.Q THEN

                eState := E_SequenceState.SEQ_DOSING;

            END_IF;



        // -------------------------------------------------
        // DOSING / SCREW RETURN
        // -------------------------------------------------

        E_SequenceState.SEQ_DOSING:

            bRotateCmd := TRUE;

            // Continue dosing until screw reaches rear position.

            IF bAtRear THEN

                bRotateCmd := FALSE;

                eState := E_SequenceState.SEQ_OPEN_MOLD;

            END_IF;



        // -------------------------------------------------
        // OPEN MOLD
        // -------------------------------------------------

        E_SequenceState.SEQ_OPEN_MOLD:

            bOpenMoldCmd := TRUE;

            IF bMoldOpen THEN

                bOpenMoldCmd := FALSE;

                eState := E_SequenceState.SEQ_EJECT;

            END_IF;



        // -------------------------------------------------
        // PART EJECTION
        // -------------------------------------------------

        E_SequenceState.SEQ_EJECT:

            // Part has physically completed the molding process.
            // MAIN uses this pulse to increment TotalParts.

            bPartCompleted := TRUE;

            // Newly produced part must now be inspected.

            eState := E_SequenceState.SEQ_VISION_TRIGGER;



        // -------------------------------------------------
        // VISION TRIGGER
        // -------------------------------------------------

        E_SequenceState.SEQ_VISION_TRIGGER:

            // Camera unavailable before inspection.
            // Current part cannot be verified, therefore reject
            // it and request a graceful machine stop.

            IF bVisionOffline OR bVisionTimeout THEN

                bRejectedPart := TRUE;

                bStopLatched := TRUE;

                eState := E_SequenceState.SEQ_CLOSE_MOLD;


            // Camera available and ready.

            ELSIF bVisionReady THEN

                // One-scan trigger pulse.

                bVisionTrigger := TRUE;

                eState := E_SequenceState.SEQ_VISION_WAIT;

            END_IF;



        // -------------------------------------------------
        // WAIT FOR VISION RESULT
        // -------------------------------------------------

        E_SequenceState.SEQ_VISION_WAIT:

            // Communication failure or inspection timeout
            // while waiting for result.

            IF bVisionOffline OR bVisionTimeout THEN

                // Treat unverified part as rejected.

                bRejectedPart := TRUE;

                // Finish safely and stop production.

                bStopLatched := TRUE;

                eState := E_SequenceState.SEQ_CLOSE_MOLD;


            // Normal inspection completed.

            ELSIF bVisionResultValid THEN

                eState := E_SequenceState.SEQ_SORT_PART;

            END_IF;



        // -------------------------------------------------
        // SORT / CLASSIFY PART
        // -------------------------------------------------

        E_SequenceState.SEQ_SORT_PART:

            IF bVisionPartOK THEN

                bGoodPart := TRUE;

            ELSE

                bRejectedPart := TRUE;

            END_IF;


            // Tell vision system that PLC has consumed result.

            bVisionAck := TRUE;


            // Continue machine cycle.

            eState := E_SequenceState.SEQ_CLOSE_MOLD;



        // -------------------------------------------------
        // CLOSE MOLD
        // -------------------------------------------------

        E_SequenceState.SEQ_CLOSE_MOLD:

            bCloseMoldCmd := TRUE;

            IF bMoldClosed THEN

                bCloseMoldCmd := FALSE;
				
				// Complete cycle time includes vision inspection
        		tLastCycleTime := fbCycleTimer.ET;

        		// Stop/reset timer before next cycle
        		bCycleTiming := FALSE;

                eState := E_SequenceState.SEQ_COMPLETE;

            END_IF;



        // -------------------------------------------------
        // CYCLE COMPLETE
        // -------------------------------------------------

        E_SequenceState.SEQ_COMPLETE:

            // Graceful stop requested or production batch complete.

            IF bStopLatched
               OR (nProducedParts >= nBatchSize) THEN

                bStopComplete := TRUE;

                eState := E_SequenceState.SEQ_IDLE;


            // Otherwise immediately start next product.

            ELSE

				// Start timing the next production cycle
    			bCycleTiming := TRUE;			
                eState := E_SequenceState.SEQ_INJECT;

            END_IF;



        // -------------------------------------------------
        // FALLBACK
        // -------------------------------------------------

        ELSE

            eState := E_SequenceState.SEQ_IDLE;

    END_CASE;

END_IF;

END_FUNCTION_BLOCK

// ---- POUs/FB_Extruder.TcPOU
FUNCTION_BLOCK FB_Extruder
VAR_INPUT
	bRotateCmd		:  BOOL;
	bInjectCmd		:  BOOL;
	
	bES101			:  BOOL;
	bES102			:  BOOL;
END_VAR
VAR_OUTPUT
	bRotateRequest	:  BOOL;
	bInjectRequest  :  BOOL;
	
	bAtFront		:  BOOL;
	bAtRear			:  BOOL;
	bBusy			:  BOOL;
	
	bCommandConflict:  BOOL;
END_VAR
VAR
END_VAR

// Screw position
bAtFront := bES101;
bAtRear  := bES102;

// M101 and M102 must never be requested together
bCommandConflict :=
    bRotateCmd AND bInjectCmd;

// Rotation / dosing request
bRotateRequest :=
    bRotateCmd
    AND NOT bInjectCmd;

// Injection request
bInjectRequest :=
    bInjectCmd
    AND NOT bRotateCmd
    AND NOT bAtFront;

// Equipment busy
bBusy :=
    bRotateRequest OR bInjectRequest;

END_FUNCTION_BLOCK

// ---- POUs/FB_Mold.TcPOU
FUNCTION_BLOCK FB_Mold
VAR_INPUT
	bOpenCmd		:  BOOL;
	bCloseCmd		:  BOOL;
	
	bES201			:  BOOL;
	bES202			:  BOOL;
END_VAR
VAR_OUTPUT
	bOpenRequest	:  BOOL;
	bCloseRequest	:  BOOL;
	
	bIsOpen			:  BOOL;
	bIsClosed		:  BOOL;
	bMoving			:  BOOL;
	
	bCommandConflict:  BOOL;
END_VAR
VAR
END_VAR

// Position status
bIsOpen   := bES201;
bIsClosed := bES202;

// Detect contradictory commands
bCommandConflict :=
    bOpenCmd AND bCloseCmd;

// Generate requests
bOpenRequest :=
    bOpenCmd
    AND NOT bCloseCmd
    AND NOT bIsOpen;

bCloseRequest :=
    bCloseCmd
    AND NOT bOpenCmd
    AND NOT bIsClosed;

// Motion status
bMoving :=
    bOpenRequest OR bCloseRequest;

END_FUNCTION_BLOCK

// ---- POUs/FB_Hopper.TcPOU
FUNCTION_BLOCK FB_Hopper
VAR_INPUT
	eMode			: E_MachineMode;
	
	bLIS101			: BOOL;
	bLIS102			: BOOL;
	
	bAck			: BOOL;
END_VAR
VAR_OUTPUT
	bFeederRequest	: BOOL;
	bWarning		: BOOL;
	bRefilling		: BOOL;
	
	bLowLevelTimeout	: BOOL;
	bFillTimeout	: BOOL;
END_VAR
VAR
	fbLowLevelTimer	: TON;
	fbFIllTimer		: TON;
	
	bAutoEnabled	: BOOL;
END_VAR

								// Automatic refill is allowed only during
									// STARTUP or normal RUN operati
								
bAutoEnabled := (eMode = E_MachineMode.MODE_STARTUP) OR (eMode = E_MachineMode.MODE_RUN);

//Warning Acknowledgement

IF bAck THEN
	bWarning := FALSE;
	bLowLevelTimeout := FALSE;
    bFillTimeout := FALSE;
END_IF

//Start Auto Refill

IF bAutoEnabled
	AND NOT bWarning
	AND NOT bLIS101
	AND NOT bRefilling THEN
		bRefilling := TRUE;
END_IF;

//Stop when high level is reached

IF bLIS102 THEN
    bRefilling := FALSE;
END_IF;

// Stop refilling outside permitted machine modes
IF NOT bAutoEnabled THEN
    bRefilling := FALSE;
END_IF;

// Timer 1:
// Low-level switch must recover within 30 seconds

fbLowLevelTimer(
	IN := bRefilling AND NOT bLIS101,
	PT := GVL_Config.c_tHopperLowTimeout
);

IF fbLowLevelTimer.Q THEN
    bLowLevelTimeout := TRUE;
END_IF;

// Timer 2:
// Complete filling must finish within 180 seconds

fbFillTimer(
    IN := bRefilling,
    PT := GVL_Config.c_tHopperFillTimeout
);

IF fbFillTimer.Q THEN
    bFillTimeout := TRUE;
END_IF;

// Fault handling

IF bLowLevelTimeout OR bFillTimeout THEN

    bWarning := TRUE;
    bRefilling := FALSE;

END_IF;

// Feeder motor request

bFeederRequest :=
    bRefilling
    AND bAutoEnabled
    AND NOT bWarning;

END_FUNCTION_BLOCK

// ---- POUs/FB_AlarmManager.TcPOU
FUNCTION_BLOCK FB_AlarmManager
VAR_INPUT
    eMode : E_MachineMode;

    // Hopper
    bHopperLowTimeout  : BOOL;
    bHopperFillTimeout : BOOL;

    // Process
    fBarrelTemp  : REAL;
    fPressureBar : REAL;

    // Safety / machine
    bGuardOpen : BOOL;
    bEStop     : BOOL;

    // Vision - used later
    bVisionOffline : BOOL;
    bVisionTimeout : BOOL;

    // Operator
    bAck : BOOL;
END_VAR

VAR_OUTPUT
    bFaultActive : BOOL;
    eActiveAlarm : E_AlarmID := E_AlarmID.ALARM_NONE;
END_VAR

// Default

bFaultActive := FALSE;
eActiveAlarm := E_AlarmID.ALARM_NONE;

// Alarm priority
// Highest priority first


// Emergency Stop
IF bEStop THEN

    bFaultActive := TRUE;
    eActiveAlarm := E_AlarmID.ALARM_ESTOP;
	

// High pressure
ELSIF fPressureBar > GVL_Config.c_fMaxPressure THEN

    bFaultActive := TRUE;
    eActiveAlarm := E_AlarmID.ALARM_PRESSURE_HIGH;


// Guard opened during active machine operation
ELSIF bGuardOpen
      AND (
          (eMode = E_MachineMode.MODE_STARTUP)
          OR
          (eMode = E_MachineMode.MODE_RUN)
      ) THEN

    bFaultActive := TRUE;
    eActiveAlarm := E_AlarmID.ALARM_GUARD_OPEN;


// Hopper low-level timeout
ELSIF bHopperLowTimeout THEN

    bFaultActive := TRUE;
    eActiveAlarm := E_AlarmID.ALARM_HOPPER_LOW_TIMEOUT;


// Hopper full-level timeout
ELSIF bHopperFillTimeout THEN

    bFaultActive := TRUE;
    eActiveAlarm := E_AlarmID.ALARM_HOPPER_FILL_TIMEOUT;

// Vision communication fault
ELSIF bVisionOffline THEN

    bFaultActive := TRUE;
    eActiveAlarm := E_AlarmID.ALARM_VISION_OFFLINE;


// Vision result timeout
ELSIF bVisionTimeout THEN

    bFaultActive := TRUE;
    eActiveAlarm := E_AlarmID.ALARM_VISION_TIMEOUT;

END_IF;

END_FUNCTION_BLOCK

// ---- POUs/FB_Interlocks.TcPOU
FUNCTION_BLOCK FB_Interlocks
VAR_INPUT
	// Requested actuator commands
    eMode			: E_MachineMode;
	
	bM101_Request   : BOOL;
    bM102_Request   : BOOL;
    bM201_l_Request : BOOL;
    bM201_r_Request : BOOL;

    // Sensors
    bES101          : BOOL;
    bES102          : BOOL;
    bES201          : BOOL;
    bES202          : BOOL;

    bGuardOpen      : BOOL;

    // Process values
    fPressureBar    : REAL;
    fBarrelTemp     : REAL;
END_VAR
VAR_OUTPUT
	// Safe actuator commands
    bM101_Enable    : BOOL;
    bM102_Enable    : BOOL;
    bM201_l_Enable  : BOOL;
    bM201_r_Enable  : BOOL;

	// Status
    bPressureOK     : BOOL;
    bTemperatureOK  : BOOL;
    bGuardOK        : BOOL;
END_VAR
VAR
END_VAR


											// Basic permissives

bPressureOK :=
    fPressureBar <= GVL_Config.c_fMaxPressure;

bTemperatureOK :=
    fBarrelTemp >= GVL_Config.c_fMinOperatingTemp;

bGuardOK :=
    NOT bGuardOpen;

										// M101 - Extruder screw rotation

bM101_Enable :=
    bM101_Request
    AND bPressureOK
    AND bTemperatureOK
    AND NOT bM102_Request
	AND
	(
		(eMode = E_MachineMode.MODE_STARTUP)
		OR NOT bES102
	);
	
											// M102 - Injection cylinder

bM102_Enable :=
    bM102_Request
    AND bGuardOK
    AND bPressureOK
    AND bTemperatureOK
    AND NOT bES101
    AND NOT bM101_Request;

													// Mold opening

bM201_l_Enable :=
    bM201_l_Request
    AND bGuardOK
    AND NOT bES201
    AND NOT bM201_r_Request;

													// Mold closing

bM201_r_Enable :=
    bM201_r_Request
    AND bGuardOK
    AND NOT bES202
    AND NOT bM201_l_Request;

END_FUNCTION_BLOCK

// ---- POUs/FB_Vision.TcPOU
FUNCTION_BLOCK FB_Vision
VAR_INPUT
    // Machine / handshake
    bEnable       : BOOL;
    bTrigger      : BOOL;
    bAck          : BOOL;
    bFaultAck     : BOOL;

    // Simulation of technical faults
    bForceOffline : BOOL;
    bForceTimeout : BOOL;

    // Current product
    nProductID    : DINT;

    // Software-in-the-loop image source
    sImagePath    : STRING(255);
END_VAR


VAR_OUTPUT
    stResult : ST_VisionResult;

    bOffline : BOOL;
    bTimeout : BOOL;
    bError   : BOOL;
END_VAR


VAR
    // =================================================
    // HANDSHAKE / STATE MACHINE
    // =================================================

    fbTrigger      : R_TRIG;
    fbTimeoutTimer : TON;

    nState : USINT := 0;

    bReadCmd          : BOOL := FALSE;
    bInspectionActive : BOOL := FALSE;

    sActiveImagePath : STRING(255);
    nActiveProductID : DINT := 0;


    // =================================================
    // IMAGE ACQUISITION
    // =================================================

    fbReadImage : FB_VN_ReadImage;

    ipImageIn : ITcVnImage;

    nReadErrorId : UDINT := 0;


    // =================================================
    // IMAGE PROCESSING
    // =================================================

    ipImageGray   : ITcVnImage;
    ipImageBinary : ITcVnImage;
    ipPartMask    : ITcVnImage;

    hrVision : HRESULT := S_OK;

    nImageWidth  : UDINT := 0;
    nImageHeight : UDINT := 0;

    fThreshold : LREAL := 128.0;


    // =================================================
    // HOLE ANALYSIS
    // =================================================

    ipLabelImage    : ITcVnImage;
    ipBoundingBoxes : ITcVnContainer;
    ipNumPixels     : ITcVnContainer;
    ipCentroids     : ITcVnContainer;

    nLabels : DINT := 0;

    nPixels0 : DINT := 0;
    nPixels1 : DINT := 0;
    nPixels2 : DINT := 0;
    nPixels3 : DINT := 0;

    fHoleAreaDifferencePct : LREAL := 100.0;

    bHoleCountOK : BOOL := FALSE;
    bHoleSizeOK  : BOOL := FALSE;


    // =================================================
    // PART GEOMETRY
    // =================================================

    ipPartLabelImage    : ITcVnImage;
    ipPartBoundingBoxes : ITcVnContainer;
    ipPartNumPixels     : ITcVnContainer;
    ipPartCentroids     : ITcVnContainer;

    nPartLabels : DINT := 0;
    nPartPixels : DINT := 0;

    stPartBox : TcVnRectangle_DINT;

    bWidthOK    : BOOL := FALSE;
    bHeightOK   : BOOL := FALSE;
    bPartAreaOK : BOOL := FALSE;
    bShapeOK    : BOOL := FALSE;


    // =================================================
    // LOCAL ROI INSPECTION
    // =================================================

    ipCornerROI : ITcVnImage;
    ipNotchROI  : ITcVnImage;

    nCornerPixels : ULINT := 0;
    nNotchPixels  : ULINT := 0;

    nRefCornerPixels : ULINT := 4539;
    nRefNotchPixels  : ULINT := 10400;

    fCornerDifferencePct : LREAL := 100.0;
    fNotchDifferencePct  : LREAL := 100.0;

    bCornerOK : BOOL := FALSE;
    bNotchOK  : BOOL := FALSE;


    // =================================================
    // FINAL INSPECTION
    // =================================================

    bInspectionOK : BOOL := FALSE;


    // =================================================
    // ADS IMAGE WATCH
    // =================================================

    ipImageDisplay    : ITcVnDisplayableImage;
    ipGrayDisplay     : ITcVnDisplayableImage;
    ipBinaryDisplay   : ITcVnDisplayableImage;
    ipPartMaskDisplay : ITcVnDisplayableImage;
END_VAR

// =====================================================
// VISION STATE MACHINE
// =====================================================


// -----------------------------------------------------
// Trigger edge
// -----------------------------------------------------

fbTrigger(CLK := bTrigger);


// -----------------------------------------------------
// Communication state
// -----------------------------------------------------

bOffline := bForceOffline;


// Read command is a one-scan pulse
bReadCmd := FALSE;


// -----------------------------------------------------
// Fault acknowledgement
// -----------------------------------------------------

IF bFaultAck AND NOT bOffline THEN

    bTimeout := FALSE;
    bError := FALSE;

    IF nState = 90 THEN
        nState := 0;
    END_IF;

END_IF;


// -----------------------------------------------------
// Camera / vision offline
// -----------------------------------------------------

IF bOffline THEN

    stResult.bResultValid := FALSE;

    nState := 90;

END_IF;


// =====================================================
// MAIN VISION STATE MACHINE
// =====================================================

CASE nState OF


    // =================================================
    // 0 - IDLE / READY
    // =================================================

    0:

        IF bEnable
           AND NOT bOffline
           AND NOT bTimeout
           AND NOT bError
           AND fbTrigger.Q THEN

            // Capture the values associated with this part.

            sActiveImagePath := sImagePath;
            nActiveProductID := nProductID;

			nReadErrorId := 0;
			
            // Clear previous result.

            stResult.bResultValid := FALSE;
            stResult.bPartPresent := FALSE;
            stResult.bPartOK := FALSE;

            stResult.nDefectCode := UINT#0;

            stResult.fWidth := 0.0;
            stResult.fHeight := 0.0;
            stResult.fAngle := 0.0;

            stResult.nProductID := nActiveProductID;


            // Begin acquisition.

            nState := 10;

        END_IF;



    // =================================================
    // 10 - START IMAGE READ
    // =================================================

    10:

        // Generate one-scan rising edge for FB_VN_ReadImage.

        bReadCmd := TRUE;

        nState := 20;



    // =================================================
    // 20 - WAIT FOR IMAGE
    // =================================================

    20:

        // Image-reading error

        IF fbReadImage.bError THEN

            nReadErrorId := fbReadImage.nErrorId;

            bError := TRUE;

            // Image load / acquisition error
            stResult.nDefectCode := UINT#401;

            nState := 90;


        // Force-timeout is deliberately used during
        // commissioning to prevent progress.

        ELSIF NOT bForceTimeout
              AND NOT fbReadImage.bBusy
              AND (ipImageIn <> 0) THEN

            nState := 30;

        END_IF;
		
	
		// =================================================
    	// 30 - PROCESS IMAGE
    	// =================================================

	30:

        hrVision := S_OK;

        bInspectionOK := FALSE;

        bHoleCountOK := FALSE;
        bHoleSizeOK := FALSE;

        bWidthOK := FALSE;
        bHeightOK := FALSE;
        bPartAreaOK := FALSE;
        bShapeOK := FALSE;

        bCornerOK := FALSE;
        bNotchOK := FALSE;

        nPixels0 := 0;
        nPixels1 := 0;
        nPixels2 := 0;
        nPixels3 := 0;

        nPartPixels := 0;

        fHoleAreaDifferencePct := 100.0;
        fCornerDifferencePct := 100.0;
        fNotchDifferencePct := 100.0;
		
		// =================================================
    	// 1. IMAGE DIMENSIONS
    	// =================================================

    	hrVision := F_VN_GetImageWidth(
        	ipImageIn,
        	nImageWidth,
        	hrVision
    	);

    	hrVision := F_VN_GetImageHeight(
        	ipImageIn,
        	nImageHeight,
        	hrVision
    	);


    	// =================================================
    	// 2. COLOR -> GRAYSCALE
    	// =================================================

   		hrVision := F_VN_ConvertColorSpace(
        	ipSrcImage := ipImageIn,
        	ipDestImage := ipImageGray,
        	eTransform := TCVN_CST_BGR_TO_GRAY,
        	hrPrev := hrVision
    	);


    	// =================================================
    	// 3. NORMAL BINARY MASK
    	//
    	// Background = WHITE
    	// Holes      = WHITE
    	// Part       = BLACK
    	// =================================================

    	hrVision := F_VN_Threshold(
        	ipSrcImage := ipImageGray,
        	ipDestImage := ipImageBinary,
        	fThreshold := fThreshold,
        	fMaxValue := 255.0,
        	eThresholdType := TCVN_TT_BINARY,
        	hrPrev := hrVision
    	);


    	// =================================================
    	// 4. INVERTED PART MASK
    	//
    	// Part       = WHITE
    	// Background = BLACK
    	// Holes      = BLACK
    	// =================================================

    	hrVision := F_VN_Threshold(
        	ipSrcImage := ipImageGray,
        	ipDestImage := ipPartMask,
        	fThreshold := fThreshold,
        	fMaxValue := 255.0,
        	eThresholdType := TCVN_TT_BINARY_INV,
        	hrPrev := hrVision
    	);
	

    	// =================================================
    	// 5. LOCAL ROI INSPECTION
    	// =================================================


    	// -------------------------------------------------
    	// TOP-RIGHT CORNER ROI
    	// Detect chipped corner
    	// -------------------------------------------------

    	hrVision := F_VN_CopyImageRegion(
        	ipSrcImage := ipPartMask,
        	nX := 970,
        	nY := 245,
        	nWidth := 100,
        	nHeight := 60,
        	ipDestImage := ipCornerROI,
        	hrPrev := hrVision
    	);

    	hrVision := F_VN_CountNonZeroPixels(
        	ipSrcImage := ipCornerROI,
        	nNonZero := nCornerPixels,
        	hrPrev := hrVision
    	);


    	// -------------------------------------------------
    	// BOTTOM-CENTER NOTCH ROI
    	// Detect malformed notch
    	// -------------------------------------------------

    	hrVision := F_VN_CopyImageRegion(
        	ipSrcImage := ipPartMask,
        	nX := 640,
        	nY := 680,
        	nWidth := 170,
        	nHeight := 148,
        	ipDestImage := ipNotchROI,
        	hrPrev := hrVision
    	);

    	hrVision := F_VN_CountNonZeroPixels(
        	ipSrcImage := ipNotchROI,
        	nNonZero := nNotchPixels,
        	hrPrev := hrVision
    	);


    	// =================================================
    	// 6. OUTER PART GEOMETRY
    	// =================================================

    	hrVision := F_VN_ConnectedComponentsWithStats(
        	ipSrcImage := ipPartMask,
        	ipLabelImage := ipPartLabelImage,
        	ipBoundingBoxes := ipPartBoundingBoxes,
        	ipNumPixels := ipPartNumPixels,
        	ipCentroids := ipPartCentroids,
        	nLabels := nPartLabels,
        	hrPrev := hrVision
    	);


    	// Expected:
    	//
    	// label 0 = black background
    	// label 1 = white molded part

    	IF nPartLabels >= 2 THEN

        	hrVision := F_VN_GetAt_DINT(
            	ipContainer := ipPartNumPixels,
            	nElement := nPartPixels,
            	nIndex := 1,
            	hrPrev := hrVision
        	);

        	hrVision := F_VN_GetAt_TcVnRectangle_DINT(
            	ipContainer := ipPartBoundingBoxes,
            	stElement := stPartBox,
            	nIndex := 1,
            	hrPrev := hrVision
        	);


        	// ---------------------------------------------
        	// Width check
        	//
        	// Reference = 672 px
        	// Approximately +/- 3 %
        	// ---------------------------------------------

        	bWidthOK :=
            	(stPartBox.nWidth >= 652)
            	AND
            	(stPartBox.nWidth <= 692);


        	// ---------------------------------------------
        	// Height check
        	//
        	// Reference = 577 px
        	// Approximately +/- 3 %
        	// ---------------------------------------------

        	bHeightOK :=
            	(stPartBox.nHeight >= 560)
            	AND
            	(stPartBox.nHeight <= 594);


        	// ---------------------------------------------
        	// Part-area check
        	//
        	// Reference = 350970 px
        	// Approximately +/- 3 %
        	// ---------------------------------------------

        	bPartAreaOK :=
            	(nPartPixels >= 340441)
            	AND
            	(nPartPixels <= 361499);

    	ELSE

        	// Part could not be identified

        	bWidthOK := FALSE;
        	bHeightOK := FALSE;
        	bPartAreaOK := FALSE;

    	END_IF;


    	// Overall global shape check

    	bShapeOK :=
        	bWidthOK
        	AND
        	bHeightOK
        	AND
        	bPartAreaOK;


    	// =================================================
    	// 7. HOLE ANALYSIS
    	// =================================================

    	hrVision := F_VN_ConnectedComponentsWithStats(
        	ipSrcImage := ipImageBinary,
        	ipLabelImage := ipLabelImage,
        	ipBoundingBoxes := ipBoundingBoxes,
        	ipNumPixels := ipNumPixels,
        	ipCentroids := ipCentroids,
        	nLabels := nLabels,
        	hrPrev := hrVision
    	);


    	// -------------------------------------------------
    	// Safely extract components
    	// -------------------------------------------------

    	IF nLabels >= 1 THEN

        	hrVision := F_VN_GetAt_DINT(
            	ipContainer := ipNumPixels,
            	nElement := nPixels0,
            	nIndex := 0,
            	hrPrev := hrVision
        	);

    	END_IF;


    	IF nLabels >= 2 THEN

        	hrVision := F_VN_GetAt_DINT(
            	ipContainer := ipNumPixels,
            	nElement := nPixels1,
            	nIndex := 1,
            	hrPrev := hrVision
        	);

    	END_IF;


    	IF nLabels >= 3 THEN

        	hrVision := F_VN_GetAt_DINT(
            	ipContainer := ipNumPixels,
            	nElement := nPixels2,
            	nIndex := 2,
            	hrPrev := hrVision
        	);

    	END_IF;


    	IF nLabels >= 4 THEN

        	hrVision := F_VN_GetAt_DINT(
            	ipContainer := ipNumPixels,
            	nElement := nPixels3,
            	nIndex := 3,
            	hrPrev := hrVision
        	);

    	END_IF;


    	// -------------------------------------------------
    	// Hole-count check
    	//
    	// Good image:
    	//
    	// label 0 = black part
    	// label 1 = outside white background
    	// label 2 = hole 1
    	// label 3 = hole 2
    	//
    	// Therefore expected nLabels = 4
    	// -------------------------------------------------

    	bHoleCountOK := (nLabels = 4);


    	// -------------------------------------------------
    	// Hole-size comparison
    	// -------------------------------------------------

    	IF bHoleCountOK
       	AND (nPixels2 > 0)
       	AND (nPixels3 > 0) THEN

        	fHoleAreaDifferencePct :=
            	ABS(
                	DINT_TO_LREAL(
                    	nPixels2 - nPixels3
                	)
            	)
            	/
            	DINT_TO_LREAL(
                	MAX(nPixels2, nPixels3)
            	)
            	* 100.0;


        	// Maximum difference = 10 %

        	bHoleSizeOK :=
            	fHoleAreaDifferencePct <= 10.0;

    	ELSE

        	fHoleAreaDifferencePct := 100.0;
        	bHoleSizeOK := FALSE;

    	END_IF;


    	// =================================================
    	// 8. CORNER ROI CHECK
    	// =================================================

    	// Reference from deterministic good image:
    	//
    	// nRefCornerPixels = 4539

    	IF nRefCornerPixels > 0 THEN

        	IF nCornerPixels >= nRefCornerPixels THEN

            	fCornerDifferencePct :=
                	ULINT_TO_LREAL(
                    	nCornerPixels - nRefCornerPixels
                	)
                	/
                	ULINT_TO_LREAL(
                    	nRefCornerPixels
                	)
                	* 100.0;

        	ELSE

            	fCornerDifferencePct :=
                	ULINT_TO_LREAL(
                    	nRefCornerPixels - nCornerPixels
                	)
                	/
                	ULINT_TO_LREAL(
                    	nRefCornerPixels
                	)
                	* 100.0;

        	END_IF;


        	// Maximum deviation = 10 %

        	bCornerOK :=
            	fCornerDifferencePct <= 10.0;

    	ELSE

        	bCornerOK := FALSE;

    	END_IF;


    	// =================================================
    	// 9. NOTCH ROI CHECK
    	// =================================================

    	// Reference from deterministic good image:
    	//
    	// nRefNotchPixels = 10400

    	IF nRefNotchPixels > 0 THEN

        	IF nNotchPixels >= nRefNotchPixels THEN

            	fNotchDifferencePct :=
                	ULINT_TO_LREAL(
                    	nNotchPixels - nRefNotchPixels
                	)
                	/
                	ULINT_TO_LREAL(
                    	nRefNotchPixels
                	)
                	* 100.0;

        	ELSE

            	fNotchDifferencePct :=
                	ULINT_TO_LREAL(
                    	nRefNotchPixels - nNotchPixels
                	)
                	/
                	ULINT_TO_LREAL(
                    	nRefNotchPixels
                	)
                	* 100.0;

        	END_IF;


        	// Maximum deviation = 10 %

        	bNotchOK :=
            	fNotchDifferencePct <= 10.0;

    	ELSE

        	bNotchOK := FALSE;

    	END_IF;


    	// =================================================
    	// 10. FINAL INSPECTION RESULT
    	//
    	// IMPORTANT:
    	// This MUST come after ALL individual checks.
    	// =================================================

    	bInspectionOK :=
        	bShapeOK
        	AND bHoleCountOK
        	AND bHoleSizeOK
        	AND bCornerOK
        	AND bNotchOK;


    	// =================================================
    	// 11. DIAGNOSTIC DISPLAY IMAGES
    	// =================================================


    	// Original

    	hrVision := F_VN_CopyIntoDisplayableImage(
        	ipSrcImage := ipImageIn,
        	ipDestImage := ipImageDisplay,
        	hrPrev := hrVision
    	);


    	// Grayscale

    	hrVision := F_VN_CopyIntoDisplayableImage(
        	ipSrcImage := ipImageGray,
        	ipDestImage := ipGrayDisplay,
        	hrPrev := hrVision
    	);


    	// Normal binary

    	hrVision := F_VN_CopyIntoDisplayableImage(
        	ipSrcImage := ipImageBinary,
        	ipDestImage := ipBinaryDisplay,
        	hrPrev := hrVision
    	);


    	// Inverted part mask

    	hrVision := F_VN_CopyIntoDisplayableImage(
        	ipSrcImage := ipPartMask,
        	ipDestImage := ipPartMaskDisplay,
        	hrPrev := hrVision
    	);



		// =====================================================
		// VISION PROCESSING SUCCESS / FAILURE
		// =====================================================

		IF hrVision = S_OK THEN

    		// ---------------------------------------------
    		// Part detected?
    		// ---------------------------------------------

    		stResult.bPartPresent :=
        		(nPartLabels >= 2);


    		// ---------------------------------------------
    		// Store measurements
    		// Currently these are pixels
    		// ---------------------------------------------

    		stResult.bPartPresent :=
    			(nPartLabels >= 2);

			IF stResult.bPartPresent THEN

    			stResult.fWidth :=
        			DINT_TO_REAL(stPartBox.nWidth);

    			stResult.fHeight :=
        			DINT_TO_REAL(stPartBox.nHeight);

			ELSE

    			stResult.fWidth := 0.0;
    			stResult.fHeight := 0.0;

			END_IF;

			stResult.fAngle := 0.0;

			stResult.nProductID :=
    			nActiveProductID;


    		// ---------------------------------------------
    		// Defect classification
    		// ---------------------------------------------

    		IF NOT stResult.bPartPresent THEN

        		stResult.nDefectCode := UINT#100;

    		ELSIF NOT bWidthOK THEN

        		stResult.nDefectCode := UINT#101;

    		ELSIF NOT bHeightOK THEN

        		stResult.nDefectCode := UINT#102;

    		ELSIF NOT bPartAreaOK THEN

        		stResult.nDefectCode := UINT#103;

    		ELSIF NOT bHoleCountOK THEN

        		stResult.nDefectCode := UINT#201;

    		ELSIF NOT bHoleSizeOK THEN

        		stResult.nDefectCode := UINT#202;

    		ELSIF NOT bCornerOK THEN

        		stResult.nDefectCode := UINT#301;

    		ELSIF NOT bNotchOK THEN

        		stResult.nDefectCode := UINT#302;

    		ELSE

        		stResult.nDefectCode := UINT#0;

    		END_IF;


    		// ---------------------------------------------
    		// Final PASS / FAIL
    		// ---------------------------------------------

    		stResult.bPartOK :=
        		bInspectionOK;


    		// Result is now available to machine sequence

    		stResult.bResultValid := TRUE;


    		// Go to RESULT HOLD state

    		nState := 40;


		ELSE

    		// ---------------------------------------------
    		// TwinCAT Vision processing error
    		// ---------------------------------------------

    		bError := TRUE;

    		stResult.bPartOK := FALSE;
    		stResult.bResultValid := FALSE;

    		stResult.nDefectCode := UINT#402;
	
    		nState := 90;

		END_IF;


	40:

    	IF bAck THEN

        	stResult.bResultValid := FALSE;

        	nState := 0;

    	END_IF;
		
	90:
    
		stResult.bResultValid := FALSE;

    	IF bFaultAck
       	AND NOT bOffline THEN

        	bTimeout := FALSE;
        	bError := FALSE;

        	nState := 0;

    	END_IF;
	
	
END_CASE;	
	

// =====================================================
// IMAGE ACQUISITION
// Must execute cyclically
// =====================================================

fbReadImage(
    sFilePath := sActiveImagePath,
    ipDestImage := ipImageIn,
    bRead := bReadCmd,
    nTimeout := T#2S
);


// =====================================================
// INSPECTION TIMEOUT
// =====================================================

bInspectionActive :=
    (nState = 10)
    OR
    (nState = 20)
    OR
    (nState = 30);


fbTimeoutTimer(
    IN := bInspectionActive,
    PT := T#5S
);


IF fbTimeoutTimer.Q THEN

    bTimeout := TRUE;

    stResult.bPartOK := FALSE;
    stResult.bResultValid := FALSE;

    // Vision inspection timeout
    stResult.nDefectCode := UINT#403;

    nState := 90;

END_IF;


// =====================================================
// HANDSHAKE STATUS
// =====================================================

// Busy while acquiring or processing image

stResult.bBusy :=
    (nState = 10)
    OR
    (nState = 20)
    OR
    (nState = 30);


// Ready only when completely idle and healthy

stResult.bReady :=
    bEnable
    AND
    (nState = 0)
    AND
    NOT bOffline
    AND
    NOT bTimeout
    AND
    NOT bError
    AND
    NOT stResult.bResultValid;

END_FUNCTION_BLOCK

// ---- POUs/PRG_VisionTest.TcPOU
PROGRAM PRG_VisionTest
VAR
    fbReadImage : FB_VN_ReadImage;

    ipImageIn : ITcVnImage;

    bReadImage : BOOL := FALSE;
    bImageLoaded : BOOL := FALSE;
    bImageError : BOOL := FALSE;

    nErrorId : UDINT := 0;
	
	// Image information
    nImageWidth  : UDINT := 0;
    nImageHeight : UDINT := 0;

    hrVision : HRESULT := S_OK;
	
	ipImageDisplay : ITcVnDisplayableImage;
	
	ipImageGray      : ITcVnImage;
	ipImageBinary    : ITcVnImage;

	ipGrayDisplay    : ITcVnDisplayableImage;
	ipBinaryDisplay  : ITcVnDisplayableImage;
	
	bProcessImage    : BOOL := FALSE;
	bProcessingDone  : BOOL := FALSE;
	fbProcessTrigger : R_TRIG;

	fThreshold       : LREAL := 128.0;
	
	ipPartMask        : ITcVnImage;
	ipPartMaskDisplay : ITcVnDisplayableImage;
	
	ipLabelImage : ITcVnImage;
	nLabels      : DINT := 0;
	
	// Connected-component statistics
	ipBoundingBoxes : ITcVnContainer;
	ipNumPixels     : ITcVnContainer;
	ipCentroids     : ITcVnContainer;

	stBox0 : TcVnRectangle_DINT;
	stBox1 : TcVnRectangle_DINT;
	stBox2 : TcVnRectangle_DINT;
	stBox3 : TcVnRectangle_DINT;

	nPixels0 : DINT := 0;
	nPixels1 : DINT := 0;
	nPixels2 : DINT := 0;
	nPixels3 : DINT := 0;
	
	bHoleCountOK : BOOL := FALSE;
	bHoleSizeOK  : BOOL := FALSE;
	bInspectionOK : BOOL := FALSE;

	fHoleAreaDifferencePct : LREAL := 0.0;
	
	// Part geometry analysis
	ipPartLabelImage    : ITcVnImage;
	ipPartBoundingBoxes : ITcVnContainer;
	ipPartNumPixels     : ITcVnContainer;
	ipPartCentroids     : ITcVnContainer;

	nPartLabels : DINT := 0;

	stPartBox    : TcVnRectangle_DINT;
	nPartPixels  : DINT := 0;
	
	// Reference geometry
	nRefWidth      : DINT := 672;
	nRefHeight     : DINT := 577;
	nRefPartPixels : DINT := 350970;

	// Inspection results
	bWidthOK    : BOOL := FALSE;
	bHeightOK   : BOOL := FALSE;
	bPartAreaOK : BOOL := FALSE;
	bShapeOK    : BOOL := FALSE;
	
	// Local ROI images
	ipCornerROI : ITcVnImage;
	ipNotchROI  : ITcVnImage;

	// Pixel counts
	nCornerPixels : ULINT := 0;
	nNotchPixels  : ULINT := 0;

	// Reference counts from good_reference.png
	nRefCornerPixels : ULINT := 4539;
	nRefNotchPixels  : ULINT := 10400;

	// Difference from reference
	fCornerDifferencePct : LREAL := 0.0;
	fNotchDifferencePct  : LREAL := 0.0;

	// Inspection results
	bCornerOK : BOOL := FALSE;
	bNotchOK  : BOOL := FALSE;
	END_VAR

// =====================================================
// READ IMAGE
// =====================================================

fbReadImage(
    sFilePath := 'C:\TcVision\defect_bad_notch.png',
    ipDestImage := ipImageIn,
    bRead := bReadImage,
    nTimeout := T#500MS
);


// -----------------------------------------------------
// New image requested
// -----------------------------------------------------

IF bReadImage THEN

    bImageLoaded := FALSE;
    bProcessingDone := FALSE;

END_IF;


// -----------------------------------------------------
// Image-read status
// -----------------------------------------------------

bImageError := fbReadImage.bError;
nErrorId := fbReadImage.nErrorId;


// -----------------------------------------------------
// Image successfully loaded
// -----------------------------------------------------

IF NOT bReadImage
   AND NOT fbReadImage.bBusy
   AND NOT fbReadImage.bError
   AND (ipImageIn <> 0) THEN

    bImageLoaded := TRUE;

END_IF;


// =====================================================
// PROCESSING TRIGGER
// =====================================================

// Must be executed every PLC scan.
// Q becomes TRUE for one scan when:
// bProcessImage FALSE -> TRUE

fbProcessTrigger(CLK := bProcessImage);


// =====================================================
// PROCESS IMAGE ONCE
// =====================================================

IF fbProcessTrigger.Q AND bImageLoaded THEN

    // -------------------------------------------------
    // Reset inspection results
    // Prevent results from previous image being reused
    // -------------------------------------------------

    bProcessingDone := FALSE;

    bHoleCountOK := FALSE;
    bHoleSizeOK := FALSE;

    bWidthOK := FALSE;
    bHeightOK := FALSE;
    bPartAreaOK := FALSE;
    bShapeOK := FALSE;

    bCornerOK := FALSE;
    bNotchOK := FALSE;

    bInspectionOK := FALSE;

    nPixels0 := 0;
    nPixels1 := 0;
    nPixels2 := 0;
    nPixels3 := 0;

    nPartPixels := 0;

    fHoleAreaDifferencePct := 100.0;
    fCornerDifferencePct := 100.0;
    fNotchDifferencePct := 100.0;

    hrVision := S_OK;


    // =================================================
    // 1. IMAGE DIMENSIONS
    // =================================================

    hrVision := F_VN_GetImageWidth(
        ipImageIn,
        nImageWidth,
        hrVision
    );

    hrVision := F_VN_GetImageHeight(
        ipImageIn,
        nImageHeight,
        hrVision
    );


    // =================================================
    // 2. COLOR -> GRAYSCALE
    // =================================================

    hrVision := F_VN_ConvertColorSpace(
        ipSrcImage := ipImageIn,
        ipDestImage := ipImageGray,
        eTransform := TCVN_CST_BGR_TO_GRAY,
        hrPrev := hrVision
    );


    // =================================================
    // 3. NORMAL BINARY MASK
    //
    // Background = WHITE
    // Holes      = WHITE
    // Part       = BLACK
    // =================================================

    hrVision := F_VN_Threshold(
        ipSrcImage := ipImageGray,
        ipDestImage := ipImageBinary,
        fThreshold := fThreshold,
        fMaxValue := 255.0,
        eThresholdType := TCVN_TT_BINARY,
        hrPrev := hrVision
    );


    // =================================================
    // 4. INVERTED PART MASK
    //
    // Part       = WHITE
    // Background = BLACK
    // Holes      = BLACK
    // =================================================

    hrVision := F_VN_Threshold(
        ipSrcImage := ipImageGray,
        ipDestImage := ipPartMask,
        fThreshold := fThreshold,
        fMaxValue := 255.0,
        eThresholdType := TCVN_TT_BINARY_INV,
        hrPrev := hrVision
    );


    // =================================================
    // 5. LOCAL ROI INSPECTION
    // =================================================


    // -------------------------------------------------
    // TOP-RIGHT CORNER ROI
    // Detect chipped corner
    // -------------------------------------------------

    hrVision := F_VN_CopyImageRegion(
        ipSrcImage := ipPartMask,
        nX := 970,
        nY := 245,
        nWidth := 100,
        nHeight := 60,
        ipDestImage := ipCornerROI,
        hrPrev := hrVision
    );

    hrVision := F_VN_CountNonZeroPixels(
        ipSrcImage := ipCornerROI,
        nNonZero := nCornerPixels,
        hrPrev := hrVision
    );


    // -------------------------------------------------
    // BOTTOM-CENTER NOTCH ROI
    // Detect malformed notch
    // -------------------------------------------------

    hrVision := F_VN_CopyImageRegion(
        ipSrcImage := ipPartMask,
        nX := 640,
        nY := 680,
        nWidth := 170,
        nHeight := 148,
        ipDestImage := ipNotchROI,
        hrPrev := hrVision
    );

    hrVision := F_VN_CountNonZeroPixels(
        ipSrcImage := ipNotchROI,
        nNonZero := nNotchPixels,
        hrPrev := hrVision
    );


    // =================================================
    // 6. OUTER PART GEOMETRY
    // =================================================

    hrVision := F_VN_ConnectedComponentsWithStats(
        ipSrcImage := ipPartMask,
        ipLabelImage := ipPartLabelImage,
        ipBoundingBoxes := ipPartBoundingBoxes,
        ipNumPixels := ipPartNumPixels,
        ipCentroids := ipPartCentroids,
        nLabels := nPartLabels,
        hrPrev := hrVision
    );


    // Expected:
    //
    // label 0 = black background
    // label 1 = white molded part

    IF nPartLabels >= 2 THEN

        hrVision := F_VN_GetAt_DINT(
            ipContainer := ipPartNumPixels,
            nElement := nPartPixels,
            nIndex := 1,
            hrPrev := hrVision
        );

        hrVision := F_VN_GetAt_TcVnRectangle_DINT(
            ipContainer := ipPartBoundingBoxes,
            stElement := stPartBox,
            nIndex := 1,
            hrPrev := hrVision
        );


        // ---------------------------------------------
        // Width check
        //
        // Reference = 672 px
        // Approximately +/- 3 %
        // ---------------------------------------------

        bWidthOK :=
            (stPartBox.nWidth >= 652)
            AND
            (stPartBox.nWidth <= 692);


        // ---------------------------------------------
        // Height check
        //
        // Reference = 577 px
        // Approximately +/- 3 %
        // ---------------------------------------------

        bHeightOK :=
            (stPartBox.nHeight >= 560)
            AND
            (stPartBox.nHeight <= 594);


        // ---------------------------------------------
        // Part-area check
        //
        // Reference = 350970 px
        // Approximately +/- 3 %
        // ---------------------------------------------

        bPartAreaOK :=
            (nPartPixels >= 340441)
            AND
            (nPartPixels <= 361499);

    ELSE

        // Part could not be identified

        bWidthOK := FALSE;
        bHeightOK := FALSE;
        bPartAreaOK := FALSE;

    END_IF;


    // Overall global shape check

    bShapeOK :=
        bWidthOK
        AND
        bHeightOK
        AND
        bPartAreaOK;


    // =================================================
    // 7. HOLE ANALYSIS
    // =================================================

    hrVision := F_VN_ConnectedComponentsWithStats(
        ipSrcImage := ipImageBinary,
        ipLabelImage := ipLabelImage,
        ipBoundingBoxes := ipBoundingBoxes,
        ipNumPixels := ipNumPixels,
        ipCentroids := ipCentroids,
        nLabels := nLabels,
        hrPrev := hrVision
    );


    // -------------------------------------------------
    // Safely extract components
    // -------------------------------------------------

    IF nLabels >= 1 THEN

        hrVision := F_VN_GetAt_DINT(
            ipContainer := ipNumPixels,
            nElement := nPixels0,
            nIndex := 0,
            hrPrev := hrVision
        );

    END_IF;


    IF nLabels >= 2 THEN

        hrVision := F_VN_GetAt_DINT(
            ipContainer := ipNumPixels,
            nElement := nPixels1,
            nIndex := 1,
            hrPrev := hrVision
        );

    END_IF;


    IF nLabels >= 3 THEN

        hrVision := F_VN_GetAt_DINT(
            ipContainer := ipNumPixels,
            nElement := nPixels2,
            nIndex := 2,
            hrPrev := hrVision
        );

    END_IF;


    IF nLabels >= 4 THEN

        hrVision := F_VN_GetAt_DINT(
            ipContainer := ipNumPixels,
            nElement := nPixels3,
            nIndex := 3,
            hrPrev := hrVision
        );

    END_IF;


    // -------------------------------------------------
    // Hole-count check
    //
    // Good image:
    //
    // label 0 = black part
    // label 1 = outside white background
    // label 2 = hole 1
    // label 3 = hole 2
    //
    // Therefore expected nLabels = 4
    // -------------------------------------------------

    bHoleCountOK := (nLabels = 4);


    // -------------------------------------------------
    // Hole-size comparison
    // -------------------------------------------------

    IF bHoleCountOK
       AND (nPixels2 > 0)
       AND (nPixels3 > 0) THEN

        fHoleAreaDifferencePct :=
            ABS(
                DINT_TO_LREAL(
                    nPixels2 - nPixels3
                )
            )
            /
            DINT_TO_LREAL(
                MAX(nPixels2, nPixels3)
            )
            * 100.0;


        // Maximum difference = 10 %

        bHoleSizeOK :=
            fHoleAreaDifferencePct <= 10.0;

    ELSE

        fHoleAreaDifferencePct := 100.0;
        bHoleSizeOK := FALSE;

    END_IF;


    // =================================================
    // 8. CORNER ROI CHECK
    // =================================================

    // Reference from deterministic good image:
    //
    // nRefCornerPixels = 4539

    IF nRefCornerPixels > 0 THEN

        IF nCornerPixels >= nRefCornerPixels THEN

            fCornerDifferencePct :=
                ULINT_TO_LREAL(
                    nCornerPixels - nRefCornerPixels
                )
                /
                ULINT_TO_LREAL(
                    nRefCornerPixels
                )
                * 100.0;

        ELSE

            fCornerDifferencePct :=
                ULINT_TO_LREAL(
                    nRefCornerPixels - nCornerPixels
                )
                /
                ULINT_TO_LREAL(
                    nRefCornerPixels
                )
                * 100.0;

        END_IF;


        // Maximum deviation = 10 %

        bCornerOK :=
            fCornerDifferencePct <= 10.0;

    ELSE

        bCornerOK := FALSE;

    END_IF;


    // =================================================
    // 9. NOTCH ROI CHECK
    // =================================================

    // Reference from deterministic good image:
    //
    // nRefNotchPixels = 10400

    IF nRefNotchPixels > 0 THEN

        IF nNotchPixels >= nRefNotchPixels THEN

            fNotchDifferencePct :=
                ULINT_TO_LREAL(
                    nNotchPixels - nRefNotchPixels
                )
                /
                ULINT_TO_LREAL(
                    nRefNotchPixels
                )
                * 100.0;

        ELSE

            fNotchDifferencePct :=
                ULINT_TO_LREAL(
                    nRefNotchPixels - nNotchPixels
                )
                /
                ULINT_TO_LREAL(
                    nRefNotchPixels
                )
                * 100.0;

        END_IF;


        // Maximum deviation = 10 %

        bNotchOK :=
            fNotchDifferencePct <= 10.0;

    ELSE

        bNotchOK := FALSE;

    END_IF;


    // =================================================
    // 10. FINAL INSPECTION RESULT
    //
    // IMPORTANT:
    // This MUST come after ALL individual checks.
    // =================================================

    bInspectionOK :=
        bShapeOK
        AND
        bHoleCountOK
        AND
        bHoleSizeOK
        AND
        bCornerOK
        AND
        bNotchOK;


    // =================================================
    // 11. DIAGNOSTIC DISPLAY IMAGES
    // =================================================


    // Original

    hrVision := F_VN_CopyIntoDisplayableImage(
        ipSrcImage := ipImageIn,
        ipDestImage := ipImageDisplay,
        hrPrev := hrVision
    );


    // Grayscale

    hrVision := F_VN_CopyIntoDisplayableImage(
        ipSrcImage := ipImageGray,
        ipDestImage := ipGrayDisplay,
        hrPrev := hrVision
    );


    // Normal binary

    hrVision := F_VN_CopyIntoDisplayableImage(
        ipSrcImage := ipImageBinary,
        ipDestImage := ipBinaryDisplay,
        hrPrev := hrVision
    );


    // Inverted part mask

    hrVision := F_VN_CopyIntoDisplayableImage(
        ipSrcImage := ipPartMask,
        ipDestImage := ipPartMaskDisplay,
        hrPrev := hrVision
    );


    // =================================================
    // 12. PROCESSING COMPLETE
    // =================================================

    IF hrVision = S_OK THEN

        bProcessingDone := TRUE;

    ELSE

        bProcessingDone := FALSE;
        bInspectionOK := FALSE;

    END_IF;

END_IF;

END_PROGRAM

// ---- GlobalTextList.TcGTLO
TEXTLIST GlobalTextList
  841 = '%.0f px'
  23 = '%.1f %%'
  319 = '%.1f bar'
  720 = '%.1f °C'
  77 = '%.1f °c'
  833 = '%.2f s'
  360 = '%d'
  617 = '%D / 40'
  345 = '%d / 40'
  375 = '%s'
  755 = '%u'
  877 = 'ACK'
  435 = 'ACTIVE'
  859 = 'ACTIVE ALARM'
  31 = 'Active Alarm:'
  975 = 'AUTOMATED QUALITY CONTROL'
  81 = 'Barrel Temperature'
  615 = 'BARREL TEMPERATURE'
  96 = 'Barrel Temperature '
  565 = 'Busy'
  661 = 'BUSY'
  72 = 'CURRENT SAMPLE'
  203 = 'Cycle Active'
  999 = 'CYCLE ACTIVE'
  247 = 'Cycle Time'
  647 = 'Defect Code'
  353 = 'DEFECT CODE\t'
  98 = 'FAIL'
  195 = 'Good Parts'
  241 = 'GOOD PARTS'
  608 = 'Height'
  514 = 'HEIGHT'
  571 = 'INJECTION PRESSURE'
  378 = 'Label'
  440 = 'Last Cycle Time'
  324 = 'LAST CYCLE TIME'
  834 = 'LAST INSPECTION'
  818 = 'LIVE PROCESS VALUES'
  184 = 'LIVE PRODUCTION DATA'
  312 = 'MACHINE MODE'
  477 = 'Machine Mode:'
  458 = 'Machine Mode::'
  967 = 'Machine Ready'
  680 = 'MACHINE READY'
  694 = 'MACHINE STATUS'
  317 = 'MEASUREMENTS'
  100 = 'Mold Temperature'
  152 = 'MOLD TEMPERATURE'
  97 = 'Part Present'
  413 = 'PART PRESENT'
  847 = 'PASS'
  296 = 'Pressure'
  566 = 'PROCESS'
  254 = 'Process Overview'
  949 = 'Product ID'
  594 = 'PRODUCT ID'
  159 = 'PRODUCTION'
  639 = 'RANDOM PART MODE'
  706 = 'Ready'
  649 = 'READY'
  722 = 'Reject Rate'
  153 = 'REJECT RATE'
  779 = 'Rejected Parts'
  130 = 'REJECTED PARTS'
  726 = 'Result'
  200 = 'RUNNING'
  269 = 'Sequence'
  525 = 'SEQUENCE\t'
  573 = 'Sequence State'
  753 = 'Sequence:'
  309 = 'SHUTDOWN'
  627 = 'SIM E-STOP'
  253 = 'SIM. E-STOP'
  723 = 'SMART INJECTION MOLDING'
  420 = 'SMART INJECTION MOLDING CELL'
  255 = 'SOFTWARE-IN-THE-LOOP  |  TwinCAT 3  |  TwinCAT Vision'
  468 = 'START'
  167 = 'STARTUP'
  198 = 'STOP'
  893 = 'SYSTEM HEALTH'
  790 = 'System Status'
  332 = 'System Status:'
  281 = 'Top Bar'
  746 = 'Total Parts'
  132 = 'TOTAL PARTS'
  45 = 'u'
  782 = 'VIRTUAL PRODUCTION SOURCE'
  399 = 'Vision & Quality'
  118 = 'Vision & QualityOverview'
  411 = 'VISION INSPECTION'
  748 = 'Vision Ready'
  885 = 'VISION STATUS'
  374 = 'Width'
  17 = 'WIDTH'
END_TEXTLIST

// ---- VISUs/Visualization_Overview.TcVIS
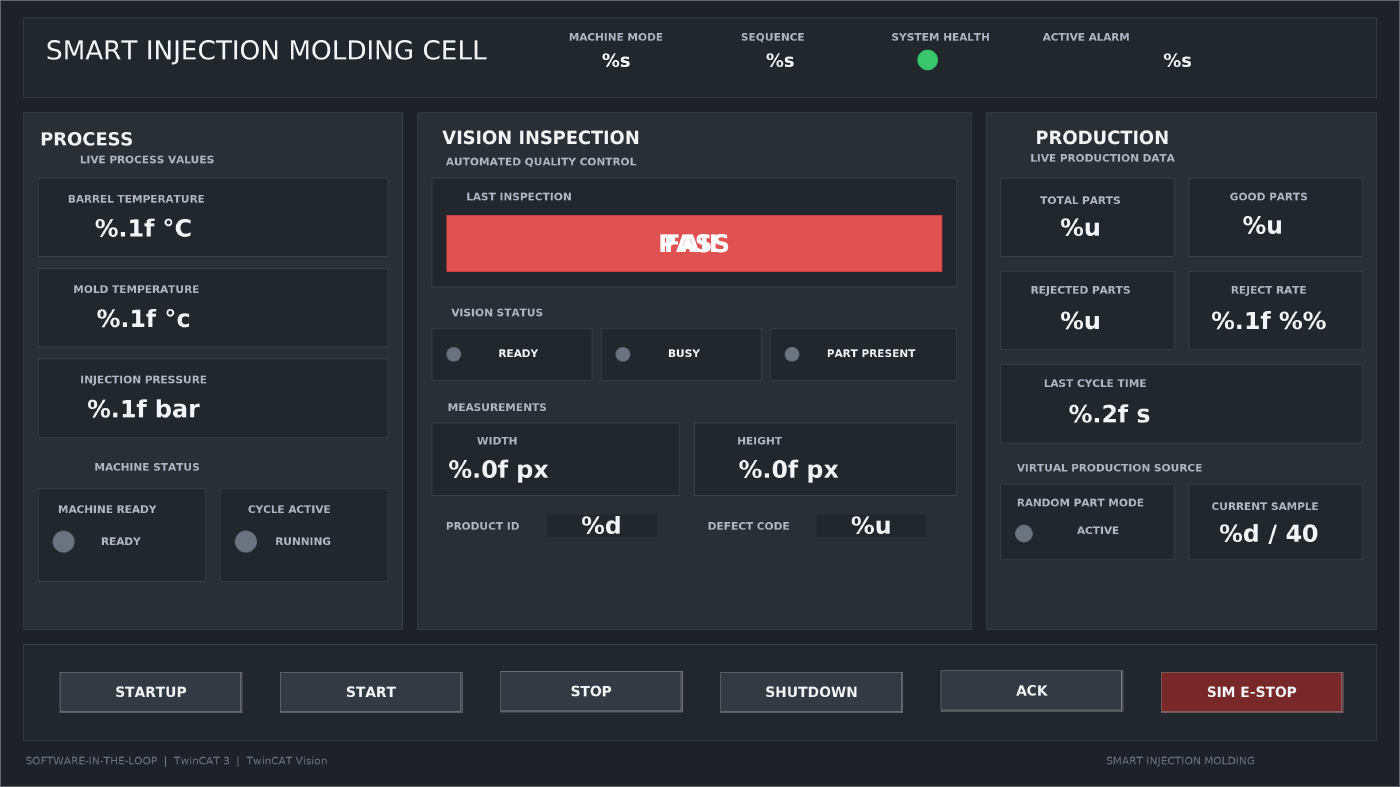
VISUALIZATION Visualization_Overview  // 1920x1080
    Rectangle (32,24 1856x110)
    Rectangle (32,154 520x710)
    Rectangle (572,154 760x710)
    Rectangle (1352,154 536x710)
    Rectangle (32,884 1856x132)
    Label (60,48 747x42), "SMART INJECTION MOLDING CELL"
    Label (760,41 170x20), "MACHINE MODE"
    Textfield (760,66 170x34), "%s", text variable: GVL_Status.sMachineModeText
    Label (960,41 210x20), "SEQUENCE"
    Textfield (960,66 220x34), "%s", text variable: GVL_Status.sSequenceText
    Label (1210,41 160x20), "SYSTEM HEALTH"
    Ellipse (1258,68 28x28), colour toggle: GVL_Status.bFaultActive
    Label (1400,41 180x20), "ACTIVE ALARM"
    Textfield (1400,66 430x34), "%s", text variable: GVL_Status.sActiveAlarmText
    Button (82,922 250x56), "STARTUP", colour toggle: GVL_IO.B_startup
        tap GVL_IO.B_startup
    Button (384,922 250x56), "START", colour toggle: GVL_IO.B_start
        tap GVL_IO.B_start
    Button (686,921 250x56), "STOP", colour toggle: GVL_IO.B_stop
        tap GVL_IO.B_stop
    Button (988,922 250x56), "SHUTDOWN", colour toggle: GVL_IO.B_shutdown
        tap GVL_IO.B_shutdown
    Button (1290,920 250x56), "ACK", colour toggle: GVL_IO.B_ack
        tap GVL_IO.B_ack
    Button (1592,922 250x56), "SIM E-STOP", colour toggle: GVL_IO.B_ES
        toggle GVL_IO.B_ES
    Label (52,174 300x34), "PROCESS"
    Label (52,208 300x22), "LIVE PROCESS VALUES"
    Rectangle (52,244 480x108)
    Label (72,262 230x22), "BARREL TEMPERATURE"
    Textfield (72,292 250x42), "%.1f °C", text variable: GVL_Status.fBarrelTemp
    Rectangle (52,368 480x108)
    Label (72,386 230x22), "MOLD TEMPERATURE"
    Textfield (72,416 250x42), "%.1f °c", text variable: GVL_Status.fMoldTemp
    Rectangle (52,492 480x108)
    Label (72,510 250x22), "INJECTION PRESSURE"
    Textfield (72,540 250x42), "%.1f bar", text variable: GVL_Status.fPressureBar
    Label (52,628 300x26), "MACHINE STATUS"
    Rectangle (52,670 230x128)
    Label (72,688 150x22), "MACHINE READY"
    Ellipse (72,728 30x30), colour toggle: GVL_Status.bMachineReady
    Label (116,730 100x26), "READY"
    Rectangle (302,670 230x128)
    Label (322,688 150x22), "CYCLE ACTIVE"
    Ellipse (322,728 30x30), colour toggle: GVL_Status.bCycleActive
    Label (366,730 100x26), "RUNNING"
    Label (592,174 300x30), "VISION INSPECTION"
    Label (592,207 300x30), "AUTOMATED QUALITY CONTROL"
    Rectangle (592,244 720x150)
    Label (612,260 200x20), "LAST INSPECTION"
    Rectangle (612,295 680x78), colour toggle: GVL_Status.stVision.bPartOK
    Label (612,295 680x78), "PASS", invisible if: NOT GVL_Status.stVision.bPartOK
    Label (612,295 680x78), "FAIL", invisible if: GVL_Status.stVision.bPartOK
    Label (592,418 180x22), "VISION STATUS"
    Rectangle (592,450 220x72)
    Ellipse (612,476 20x20), colour toggle: GVL_Status.stVision.bReady
    Label (646,470 130x30), "READY"
    Rectangle (824,450 220x72)
    Ellipse (844,476 20x20), colour toggle: GVL_Status.stVision.bBusy
    Label (878,470 120x30), "BUSY"
    Rectangle (1056,450 256x72)
    Label (1110,470 170x30), "PART PRESENT"
    Ellipse (1076,476 20x20), colour toggle: GVL_Status.stVision.bPartPresent
    Label (592,548 180x22), "MEASUREMENTS"
    Rectangle (592,580 340x100)
    Label (612,595 140x20), "WIDTH"
    Textfield (612,625 220x38), "%.0f px", text variable: GVL_Status.stVision.fWidth
    Rectangle (952,580 360x100)
    Label (972,595 140x20), "HEIGHT"
    Textfield (972,625 220x38), "%.0f px", text variable: GVL_Status.stVision.fHeight
    Label (592,710 140x24), "PRODUCT ID"
    Textfield (750,706 150x30), "%d", text variable: GVL_Status.stVision.nProductID
    Label (952,710 160x24), "DEFECT CODE"
    Textfield (1120,706 150x30), "%u", text variable: GVL_Status.stVision.nDefectCode
    Label (1372,174 280x30), "PRODUCTION"
    Label (1372,207 280x20), "LIVE PRODUCTION DATA"
    Rectangle (1372,244 238x108)
    Label (1392,260 180x30), "TOTAL PARTS"
    Textfield (1392,291 180x42), "%u", text variable: GVL_Status.stProduction.nTotalParts
    Label (1642,257 180x30), "TOTAL PARTS"
    Rectangle (1630,244 238x108)
    Textfield (1642,288 180x42), "%u", text variable: GVL_Status.stProduction.nGoodParts
    Label (1391,398 180x30), "TOTAL PARTS"
    Rectangle (1372,372 238x108)
    Textfield (1392,419 180x42), "%u", text variable: GVL_Status.stProduction.nRejectedParts
    Label (1644,401 180x30), "TOTAL PARTS"
    Rectangle (1630,372 238x108)
    Textfield (1650,419 180x42), "%.1f %%", text variable: GVL_Status.stProduction.fRejectRate
    Label (1396,724 180x30), "TOTAL PARTS"
    Rectangle (1372,664 238x104)
    Label (1650,260 180x20), "GOOD PARTS"
    Rectangle (1630,664 238x104)
    Textfield (1650,714 180x36), "%d / 40", text variable: GVL_Simulation.nVisionDatasetIndex
    Label (1392,388 180x20), "REJECTED PARTS"
    Label (1650,388 180x20), "REJECT RATE"
    Label (1392,680 180x20), "RANDOM PART MODE"
    Label (1650,680 170x30), "CURRENT SAMPLE"
    Rectangle (1372,500 496x108)
    Label (1392,516 220x20), "LAST CYCLE TIME"
    Textfield (1392,547 260x42), "%.2f s", text variable: GVL_Status.stProduction.fLastCycleTimeSec
    Label (1372,632 300x20), "VIRTUAL PRODUCTION SOURCE"
    Ellipse (1392,720 24x24), colour toggle: GVL_Simulation.bRandomPartMode
    Label (1431,713 150x30), "ACTIVE"
    Label (32,1034 900x20), "SOFTWARE-IN-THE-LOOP | TwinCAT 3 | TwinCAT Vision"
    Label (1350,1034 538x20), "SMART INJECTION MOLDING"
END_VISUALIZATION
